LIN {X 0,Y 523.661,Z 782.836,A -85,B 0,C 180,E1 -4887.396,E2 -4887.396} C_VEL
LIN {X 0,Y 523.608,Z 785.881,A -85,B 0,C 180,E1 -4887.924,E2 -4887.924} C_VEL
LIN {X 0,Y 522.919,Z 788.862,A -85,B 0,C 180,E1 -4888.477,E2 -4888.477} C_VEL
LIN {X 0,Y 519.953,Z 793.273,A -85,B 0,C 180,E1 -4889.399,E2 -4889.399} C_VEL
LIN {X 0,Y 516.983,Z 796.944,A -85,B 0,C 180,E1 -4890.367,E2 -4890.367} C_VEL
LIN {X 0,Y 516.299,Z 798.763,A -85,B 0,C 180,E1 -4890.988,E2 -4890.988} C_VEL
LIN {X 0,Y 516.19,Z 801.916,A -85,B 0,C 180,E1 -4892.422,E2 -4892.422} C_VEL
LIN {X 0,Y 516.167,Z 803.743,A -85,B 0,C 180,E1 -4893.934,E2 -4893.934} C_VEL
LIN {X 0,Y 516.163,Z 804.121,A -85,B 0,C 180,E1 -4895.221,E2 -4895.221} C_VEL
LIN {X 0,Y 516.15,Z 803.144,A -85,B 0,C 180,E1 -4896.806,E2 -4896.806} C_VEL
LIN {X 0,Y 516.166,Z 801.549,A -85,B 0,C 180,E1 -4897.843,E2 -4897.843} C_VEL
LIN {X 0,Y 516.284,Z 798.724,A -85,B 0,C 180,E1 -4899.113,E2 -4899.113} C_VEL
LIN {X 0,Y 516.35,Z 794.83,A -85,B 0,C 180,E1 -4900.342,E2 -4900.342} C_VEL
LIN {X 0,Y 516.401,Z 789.867,A -85,B 0,C 180,E1 -4901.539,E2 -4901.539} C_VEL
LIN {X 0,Y 516.631,Z 782.827,A -85,B 0,C 180,E1 -4902.857,E2 -4902.857} C_VEL
LIN {X 0,Y 516.794,Z 775.836,A -85,B 0,C 180,E1 -4903.913,E2 -4903.913} C_VEL
LIN {X 0,Y 517.07,Z 766.749,A -85,B 0,C 180,E1 -4905.028,E2 -4905.028} C_VEL
LIN {X 0,Y 517.366,Z 756.345,A -85,B 0,C 180,E1 -4906.051,E2 -4906.051} C_VEL
LIN {X 0,Y 517.663,Z 745.961,A -85,B 0,C 180,E1 -4906.873,E2 -4906.873} C_VEL
LIN {X 0,Y 517.987,Z 734.619,A -85,B 0,C 180,E1 -4907.583,E2 -4907.583} C_VEL
LIN {X 0,Y 518.283,Z 722.652,A -85,B 0,C 180,E1 -4908.16,E2 -4908.16} C_VEL
LIN {X 0,Y 518.465,Z 709.924,A -85,B 0,C 180,E1 -4908.604,E2 -4908.604} C_VEL
LIN {X 0,Y 518.673,Z 696.818,A -85,B 0,C 180,E1 -4908.89,E2 -4908.89} C_VEL
LIN {X 0,Y 518.951,Z 604.587,A -85,B 0,C 180,E1 -4910.186,E2 -4910.186} C_VEL
LIN {X 0,Y 517.134,Z 594.704,A -85,B 0,C 180,E1 -4910.404,E2 -4910.404} C_VEL
LIN {X 0,Y 517.332,Z 583.642,A -85,B 0,C 180,E1 -4912.806,E2 -4912.806} C_VEL
LIN {X 0,Y 516.951,Z 581.095,A -85,B 0,C 180,E1 -4913.399,E2 -4913.399} C_VEL
LIN {X 0,Y 516.911,Z 581.098,A -85,B 0,C 180,E1 -4916.122,E2 -4916.122} C_VEL
LIN {X 0,Y 516.887,Z 581.094,A -85,B 0,C 180,E1 -4918.937,E2 -4918.937} C_VEL
LIN {X 0,Y 516.917,Z 581.093,A -85,B 0,C 180,E1 -4921.586,E2 -4921.586} C_VEL
LIN {X 0,Y 516.929,Z 581.096,A -85,B 0,C 180,E1 -4924.212,E2 -4924.212} C_VEL
LIN {X 0,Y 516.87,Z 581.097,A -85,B 0,C 180,E1 -4926.778,E2 -4926.778} C_VEL
LIN {X 0,Y 516.938,Z 581.09,A -85,B 0,C 180,E1 -4929.732,E2 -4929.732} C_VEL
LIN {X 0,Y 516.931,Z 581.092,A -85,B 0,C 180,E1 -4932.597,E2 -4932.597} C_VEL
LIN {X 0,Y 516.942,Z 581.087,A -85,B 0,C 180,E1 -4935.031,E2 -4935.031} C_VEL
LIN {X 0,Y 517.005,Z 581.087,A -85,B 0,C 180,E1 -4938.236,E2 -4938.236} C_VEL
LIN {X 0,Y 516.969,Z 581.083,A -85,B 0,C 180,E1 -4941.401,E2 -4941.401} C_VEL
LIN {X 0,Y 517.011,Z 581.079,A -85,B 0,C 180,E1 -4943.758,E2 -4943.758} C_VEL
LIN {X 0,Y 517.086,Z 581.069,A -85,B 0,C 180,E1 -4947.664,E2 -4947.664} C_VEL
LIN {X 0,Y 517.095,Z 581.074,A -85,B 0,C 180,E1 -4950.78,E2 -4950.78} C_VEL
LIN {X 0,Y 517.016,Z 581.08,A -85,B 0,C 180,E1 -4953.118,E2 -4953.118} C_VEL
LIN {X 0,Y 517.012,Z 581.081,A -85,B 0,C 180,E1 -4956.244,E2 -4956.244} C_VEL
LIN {X 0,Y 516.957,Z 581.086,A -85,B 0,C 180,E1 -4959.39,E2 -4959.39} C_VEL
LIN {X 0,Y 516.956,Z 581.085,A -85,B 0,C 180,E1 -4961.808,E2 -4961.808} C_VEL
LIN {X 0,Y 516.948,Z 581.09,A -85,B 0,C 180,E1 -4965.147,E2 -4965.147} C_VEL
LIN {X 0,Y 516.928,Z 581.089,A -85,B 0,C 180,E1 -4968.223,E2 -4968.223} C_VEL
LIN {X 0,Y 516.916,Z 581.096,A -85,B 0,C 180,E1 -4970.702,E2 -4970.702} C_VEL
LIN {X 0,Y 516.906,Z 581.091,A -85,B 0,C 180,E1 -4974.073,E2 -4974.073} C_VEL
LIN {X 0,Y 516.93,Z 581.092,A -85,B 0,C 180,E1 -4976.658,E2 -4976.658} C_VEL
LIN {X 0,Y 516.915,Z 581.093,A -85,B 0,C 180,E1 -4979.524,E2 -4979.524} C_VEL
LIN {X 0,Y 516.899,Z 581.094,A -85,B 0,C 180,E1 -4982.544,E2 -4982.544} C_VEL
LIN {X 0,Y 516.874,Z 581.103,A -85,B 0,C 180,E1 -4985.331,E2 -4985.331} C_VEL
LIN {X 0,Y 516.885,Z 581.095,A -85,B 0,C 180,E1 -4987.944,E2 -4987.944} C_VEL
LIN {X 0,Y 516.887,Z 581.095,A -85,B 0,C 180,E1 -4990.742,E2 -4990.742} C_VEL
LIN {X 0,Y 516.886,Z 581.096,A -85,B 0,C 180,E1 -4992.832,E2 -4992.832} C_VEL
LIN {X 0,Y 516.899,Z 581.096,A -85,B 0,C 180,E1 -4995.007,E2 -4995.007} C_VEL
LIN {X 0,Y 516.919,Z 581.089,A -85,B 0,C 180,E1 -4998.399,E2 -4998.399} C_VEL
LIN {X 0,Y 516.885,Z 581.1,A -85,B 0,C 180,E1 -5001.285,E2 -5001.285} C_VEL
LIN {X 0,Y 516.875,Z 581.096,A -85,B 0,C 180,E1 -5004.22,E2 -5004.22} C_VEL
LIN {X 0,Y 516.899,Z 581.094,A -85,B 0,C 180,E1 -5007.053,E2 -5007.053} C_VEL
LIN {X 0,Y 516.897,Z 581.099,A -85,B 0,C 180,E1 -5009.797,E2 -5009.797} C_VEL
LIN {X 0,Y 516.931,Z 581.088,A -85,B 0,C 180,E1 -5012.468,E2 -5012.468} C_VEL
LIN {X 0,Y 516.88,Z 581.095,A -85,B 0,C 180,E1 -5015.07,E2 -5015.07} C_VEL
LIN {X 0,Y 516.873,Z 581.102,A -85,B 0,C 180,E1 -5017.622,E2 -5017.622} C_VEL
LIN {X 0,Y 516.936,Z 581.092,A -85,B 0,C 180,E1 -5020.13,E2 -5020.13} C_VEL
LIN {X 0,Y 516.912,Z 581.091,A -85,B 0,C 180,E1 -5022.596,E2 -5022.596} C_VEL
LIN {X 0,Y 516.948,Z 581.086,A -85,B 0,C 180,E1 -5025.03,E2 -5025.03} C_VEL
LIN {X 0,Y 516.971,Z 581.089,A -85,B 0,C 180,E1 -5028.234,E2 -5028.234} C_VEL
LIN {X 0,Y 516.97,Z 581.084,A -85,B 0,C 180,E1 -5031.4,E2 -5031.4} C_VEL
LIN {X 0,Y 517.015,Z 581.082,A -85,B 0,C 180,E1 -5033.757,E2 -5033.757} C_VEL
LIN {X 0,Y 517.089,Z 581.071,A -85,B 0,C 180,E1 -5037.663,E2 -5037.663} C_VEL
LIN {X 0,Y 517.098,Z 581.069,A -85,B 0,C 180,E1 -5040.779,E2 -5040.779} C_VEL
LIN {X 0,Y 517.017,Z 581.077,A -85,B 0,C 180,E1 -5043.117,E2 -5043.117} C_VEL
LIN {X 0,Y 517.014,Z 581.087,A -85,B 0,C 180,E1 -5046.243,E2 -5046.243} C_VEL
LIN {X 0,Y 516.95,Z 581.086,A -85,B 0,C 180,E1 -5049.389,E2 -5049.389} C_VEL
LIN {X 0,Y 516.958,Z 581.086,A -85,B 0,C 180,E1 -5051.807,E2 -5051.807} C_VEL
LIN {X 0,Y 516.95,Z 581.087,A -85,B 0,C 180,E1 -5055.146,E2 -5055.146} C_VEL
LIN {X 0,Y 516.922,Z 581.094,A -85,B 0,C 180,E1 -5058.222,E2 -5058.222} C_VEL
LIN {X 0,Y 516.918,Z 581.097,A -85,B 0,C 180,E1 -5060.701,E2 -5060.701} C_VEL
LIN {X 0,Y 516.908,Z 581.093,A -85,B 0,C 180,E1 -5064.072,E2 -5064.072} C_VEL
LIN {X 0,Y 516.929,Z 581.098,A -85,B 0,C 180,E1 -5066.658,E2 -5066.658} C_VEL
LIN {X 0,Y 516.916,Z 581.09,A -85,B 0,C 180,E1 -5069.524,E2 -5069.524} C_VEL
LIN {X 0,Y 516.901,Z 581.098,A -85,B 0,C 180,E1 -5072.543,E2 -5072.543} C_VEL
LIN {X 0,Y 516.874,Z 581.098,A -85,B 0,C 180,E1 -5075.33,E2 -5075.33} C_VEL
LIN {X 0,Y 516.886,Z 581.094,A -85,B 0,C 180,E1 -5077.943,E2 -5077.943} C_VEL
LIN {X 0,Y 516.89,Z 581.1,A -85,B 0,C 180,E1 -5080.741,E2 -5080.741} C_VEL
LIN {X 0,Y 516.89,Z 581.101,A -85,B 0,C 180,E1 -5082.831,E2 -5082.831} C_VEL
LIN {X 0,Y 516.929,Z 581.098,A -85,B 0,C 180,E1 -5085.01,E2 -5085.01} C_VEL
LIN {X 0,Y 516.919,Z 581.091,A -85,B 0,C 180,E1 -5088.398,E2 -5088.398} C_VEL
LIN {X 0,Y 516.887,Z 581.101,A -85,B 0,C 180,E1 -5091.284,E2 -5091.284} C_VEL
LIN {X 0,Y 516.878,Z 581.095,A -85,B 0,C 180,E1 -5094.219,E2 -5094.219} C_VEL
LIN {X 0,Y 516.902,Z 581.1,A -85,B 0,C 180,E1 -5097.053,E2 -5097.053} C_VEL
LIN {X 0,Y 516.892,Z 581.097,A -85,B 0,C 180,E1 -5099.796,E2 -5099.796} C_VEL
LIN {X 0,Y 516.931,Z 581.091,A -85,B 0,C 180,E1 -5102.467,E2 -5102.467} C_VEL
LIN {X 0,Y 516.962,Z 581.168,A -85,B 0,C 180,E1 -5104.186,E2 -5104.186} C_VEL
LIN {X 0,Y 518.877,Z 591.241,A -85,B 0,C 180,E1 -5105.833,E2 -5105.833} C_VEL
LIN {X 0,Y 518.458,Z 607.819,A -85,B 0,C 180,E1 -5108.321,E2 -5108.321} C_VEL
LIN {X 0,Y 517.951,Z 628.652,A -85,B 0,C 180,E1 -5111.405,E2 -5111.405} C_VEL
LIN {X 0,Y 517.414,Z 650.625,A -85,B 0,C 180,E1 -5114.621,E2 -5114.621} C_VEL
LIN {X 0,Y 519.067,Z 662.608,A -85,B 0,C 180,E1 -5114.855,E2 -5114.855} C_VEL
LIN {X 0,Y 518.619,Z 760.064,A -85,B 0,C 180,E1 -5116.231,E2 -5116.231} C_VEL
LIN {X 0,Y 518.39,Z 773.157,A -85,B 0,C 180,E1 -5116.574,E2 -5116.574} C_VEL
LIN {X 0,Y 518.11,Z 785.812,A -85,B 0,C 180,E1 -5117.066,E2 -5117.066} C_VEL
LIN {X 0,Y 517.849,Z 797.67,A -85,B 0,C 180,E1 -5117.694,E2 -5117.694} C_VEL
LIN {X 0,Y 517.502,Z 810.055,A -85,B 0,C 180,E1 -5118.543,E2 -5118.543} C_VEL
LIN {X 0,Y 517.194,Z 820.324,A -85,B 0,C 180,E1 -5119.429,E2 -5119.429} C_VEL
LIN {X 0,Y 516.94,Z 829.561,A -85,B 0,C 180,E1 -5120.412,E2 -5120.412} C_VEL
LIN {X 0,Y 516.716,Z 838.56,A -85,B 0,C 180,E1 -5121.592,E2 -5121.592} C_VEL
LIN {X 0,Y 516.511,Z 845.802,A -85,B 0,C 180,E1 -5122.769,E2 -5122.769} C_VEL
LIN {X 0,Y 516.427,Z 850.672,A -85,B 0,C 180,E1 -5123.749,E2 -5123.749} C_VEL
LIN {X 0,Y 516.314,Z 855.37,A -85,B 0,C 180,E1 -5124.923,E2 -5124.923} C_VEL
LIN {X 0,Y 516.355,Z 858.955,A -85,B 0,C 180,E1 -5126.097,E2 -5126.097} C_VEL
LIN {X 0,Y 516.283,Z 860.805,A -85,B 0,C 180,E1 -5126.878,E2 -5126.878} C_VEL
LIN {X 0,Y 516.26,Z 862.191,A -85,B 0,C 180,E1 -5127.659,E2 -5127.659} C_VEL
LIN {X 0,Y 516.16,Z 863.785,A -85,B 0,C 180,E1 -5129.219,E2 -5129.219} C_VEL
LIN {X 0,Y 516.154,Z 864,A -85,B 0,C 180,E1 -5129.999,E2 -5129.999} C_VEL
LIN {X 0,Y 516.191,Z 863.184,A -85,B 0,C 180,E1 -5131.56,E2 -5131.56} C_VEL
LIN {X 0,Y 516.26,Z 862.197,A -85,B 0,C 180,E1 -5132.34,E2 -5132.34} C_VEL
LIN {X 0,Y 516.282,Z 860.812,A -85,B 0,C 180,E1 -5133.12,E2 -5133.12} C_VEL
LIN {X 0,Y 516.344,Z 857.897,A -85,B 0,C 180,E1 -5134.292,E2 -5134.292} C_VEL
LIN {X 0,Y 516.405,Z 853.951,A -85,B 0,C 180,E1 -5135.466,E2 -5135.466} C_VEL
LIN {X 0,Y 516.479,Z 848.069,A -85,B 0,C 180,E1 -5136.797,E2 -5136.797} C_VEL
LIN {X 0,Y 516.64,Z 841.144,A -85,B 0,C 180,E1 -5138.014,E2 -5138.014} C_VEL
LIN {X 0,Y 516.844,Z 832.801,A -85,B 0,C 180,E1 -5139.193,E2 -5139.193} C_VEL
LIN {X 0,Y 517.072,Z 824.246,A -85,B 0,C 180,E1 -5140.176,E2 -5140.176} C_VEL
LIN {X 0,Y 517.432,Z 813.681,A -85,B 0,C 180,E1 -5141.159,E2 -5141.159} C_VEL
LIN {X 0,Y 517.704,Z 803.398,A -85,B 0,C 180,E1 -5141.935,E2 -5141.935} C_VEL
LIN {X 0,Y 518.016,Z 791.756,A -85,B 0,C 180,E1 -5142.636,E2 -5142.636} C_VEL
LIN {X 0,Y 518.272,Z 779.951,A -85,B 0,C 180,E1 -5143.178,E2 -5143.178} C_VEL
LIN {X 0,Y 518.472,Z 766.341,A -85,B 0,C 180,E1 -5143.621,E2 -5143.621} C_VEL
LIN {X 0,Y 518.646,Z 752.686,A -85,B 0,C 180,E1 -5143.892,E2 -5143.892} C_VEL
LIN {X 0,Y 518.905,Z 660.251,A -85,B 0,C 180,E1 -5145.177,E2 -5145.177} C_VEL
LIN {X 0,Y 517.401,Z 650.463,A -85,B 0,C 180,E1 -5145.372,E2 -5145.372} C_VEL
LIN {X 0,Y 517.889,Z 628.311,A -85,B 0,C 180,E1 -5148.596,E2 -5148.596} C_VEL
LIN {X 0,Y 518.387,Z 608.713,A -85,B 0,C 180,E1 -5151.471,E2 -5151.471} C_VEL
LIN {X 0,Y 518.791,Z 590.699,A -85,B 0,C 180,E1 -5154.165,E2 -5154.165} C_VEL
LIN {X 0,Y 516.953,Z 581.093,A -85,B 0,C 180,E1 -5155.733,E2 -5155.733} C_VEL
LIN {X 0,Y 516.918,Z 581.099,A -85,B 0,C 180,E1 -5158.414,E2 -5158.414} C_VEL
LIN {X 0,Y 516.887,Z 581.1,A -85,B 0,C 180,E1 -5161.108,E2 -5161.108} C_VEL
LIN {X 0,Y 516.91,Z 581.095,A -85,B 0,C 180,E1 -5163.966,E2 -5163.966} C_VEL
LIN {X 0,Y 516.88,Z 581.102,A -85,B 0,C 180,E1 -5166.745,E2 -5166.745} C_VEL
LIN {X 0,Y 516.9,Z 581.095,A -85,B 0,C 180,E1 -5169.718,E2 -5169.718} C_VEL
LIN {X 0,Y 516.915,Z 581.094,A -85,B 0,C 180,E1 -5171.773,E2 -5171.773} C_VEL
LIN {X 0,Y 516.918,Z 581.094,A -85,B 0,C 180,E1 -5175.009,E2 -5175.009} C_VEL
LIN {X 0,Y 516.918,Z 581.099,A -85,B 0,C 180,E1 -5178.397,E2 -5178.397} C_VEL
LIN {X 0,Y 516.904,Z 581.092,A -85,B 0,C 180,E1 -5181.286,E2 -5181.286} C_VEL
LIN {X 0,Y 516.885,Z 581.099,A -85,B 0,C 180,E1 -5184.221,E2 -5184.221} C_VEL
LIN {X 0,Y 516.892,Z 581.095,A -85,B 0,C 180,E1 -5187.053,E2 -5187.053} C_VEL
LIN {X 0,Y 516.896,Z 581.094,A -85,B 0,C 180,E1 -5189.796,E2 -5189.796} C_VEL
LIN {X 0,Y 516.923,Z 581.098,A -85,B 0,C 180,E1 -5192.467,E2 -5192.467} C_VEL
LIN {X 0,Y 516.905,Z 581.093,A -85,B 0,C 180,E1 -5195.071,E2 -5195.071} C_VEL
LIN {X 0,Y 516.879,Z 581.103,A -85,B 0,C 180,E1 -5198.462,E2 -5198.462} C_VEL
LIN {X 0,Y 516.897,Z 581.095,A -85,B 0,C 180,E1 -5200.955,E2 -5200.955} C_VEL
LIN {X 0,Y 516.908,Z 581.092,A -85,B 0,C 180,E1 -5203.41,E2 -5203.41} C_VEL
LIN {X 0,Y 516.888,Z 581.095,A -85,B 0,C 180,E1 -5205.833,E2 -5205.833} C_VEL
LIN {X 0,Y 516.996,Z 581.087,A -85,B 0,C 180,E1 -5208.234,E2 -5208.234} C_VEL
LIN {X 0,Y 516.964,Z 581.085,A -85,B 0,C 180,E1 -5211.399,E2 -5211.399} C_VEL
LIN {X 0,Y 517.002,Z 581.082,A -85,B 0,C 180,E1 -5213.757,E2 -5213.757} C_VEL
LIN {X 0,Y 517.076,Z 581.072,A -85,B 0,C 180,E1 -5217.663,E2 -5217.663} C_VEL
LIN {X 0,Y 517.087,Z 581.073,A -85,B 0,C 180,E1 -5220.779,E2 -5220.779} C_VEL
LIN {X 0,Y 517.009,Z 581.081,A -85,B 0,C 180,E1 -5223.117,E2 -5223.117} C_VEL
LIN {X 0,Y 517.007,Z 581.089,A -85,B 0,C 180,E1 -5226.243,E2 -5226.243} C_VEL
LIN {X 0,Y 516.951,Z 581.088,A -85,B 0,C 180,E1 -5229.389,E2 -5229.389} C_VEL
LIN {X 0,Y 516.975,Z 581.087,A -85,B 0,C 180,E1 -5231.824,E2 -5231.824} C_VEL
LIN {X 0,Y 516.922,Z 581.097,A -85,B 0,C 180,E1 -5235.141,E2 -5235.141} C_VEL
LIN {X 0,Y 516.987,Z 581.184,A -85,B 0,C 180,E1 -5236.638,E2 -5236.638} C_VEL
LIN {X 0,Y 517.37,Z 585.996,A -85,B 0,C 180,E1 -5237.711,E2 -5237.711} C_VEL
LIN {X 0,Y 517.11,Z 595.183,A -85,B 0,C 180,E1 -5239.708,E2 -5239.708} C_VEL
LIN {X 0,Y 519.115,Z 606.073,A -85,B 0,C 180,E1 -5239.927,E2 -5239.927} C_VEL
LIN {X 0,Y 518.62,Z 701.328,A -85,B 0,C 180,E1 -5241.28,E2 -5241.28} C_VEL
LIN {X 0,Y 518.403,Z 714.472,A -85,B 0,C 180,E1 -5241.628,E2 -5241.628} C_VEL
LIN {X 0,Y 518.174,Z 726.854,A -85,B 0,C 180,E1 -5242.109,E2 -5242.109} C_VEL
LIN {X 0,Y 517.881,Z 739.146,A -85,B 0,C 180,E1 -5242.766,E2 -5242.766} C_VEL
LIN {X 0,Y 517.582,Z 749.94,A -85,B 0,C 180,E1 -5243.507,E2 -5243.507} C_VEL
LIN {X 0,Y 517.235,Z 760.82,A -85,B 0,C 180,E1 -5244.446,E2 -5244.446} C_VEL
LIN {X 0,Y 516.994,Z 769.357,A -85,B 0,C 180,E1 -5245.354,E2 -5245.354} C_VEL
LIN {X 0,Y 516.753,Z 777.316,A -85,B 0,C 180,E1 -5246.378,E2 -5246.378} C_VEL
LIN {X 0,Y 516.575,Z 784.742,A -85,B 0,C 180,E1 -5247.553,E2 -5247.553} C_VEL
LIN {X 0,Y 516.441,Z 791.385,A -85,B 0,C 180,E1 -5248.888,E2 -5248.888} C_VEL
LIN {X 0,Y 516.32,Z 796.553,A -85,B 0,C 180,E1 -5250.241,E2 -5250.241} C_VEL
LIN {X 0,Y 516.299,Z 798.763,A -85,B 0,C 180,E1 -5250.988,E2 -5250.988} C_VEL
LIN {X 0,Y 515.62,Z 800.372,A -85,B 0,C 180,E1 -5251.615,E2 -5251.615} C_VEL
LIN {X 0,Y 512.675,Z 802.519,A -85,B 0,C 180,E1 -5252.642,E2 -5252.642} C_VEL
LIN {X 0,Y 510.201,Z 803.709,A -85,B 0,C 180,E1 -5253.48,E2 -5253.48} C_VEL
LIN {X 0,Y 509.161,Z 804.278,A -85,B 0,C 180,E1 -5254.132,E2 -5254.132} C_VEL
LIN {X 0,Y 509.09,Z 804.395,A -85,B 0,C 180,E1 -5254.354,E2 -5254.354} C_VEL
LIN {X 0,Y 509.079,Z 804.487,A -85,B 0,C 180,E1 -5255.463,E2 -5255.463} C_VEL
LIN {X 0,Y 509.063,Z 803.579,A -85,B 0,C 180,E1 -5256.802,E2 -5256.802} C_VEL
LIN {X 0,Y 509.096,Z 801.528,A -85,B 0,C 180,E1 -5258.107,E2 -5258.107} C_VEL
LIN {X 0,Y 509.228,Z 798.463,A -85,B 0,C 180,E1 -5259.41,E2 -5259.41} C_VEL
LIN {X 0,Y 509.291,Z 794.427,A -85,B 0,C 180,E1 -5260.628,E2 -5260.628} C_VEL
LIN {X 0,Y 509.38,Z 789.237,A -85,B 0,C 180,E1 -5261.839,E2 -5261.839} C_VEL
LIN {X 0,Y 509.602,Z 782.773,A -85,B 0,C 180,E1 -5263.037,E2 -5263.037} C_VEL
LIN {X 0,Y 509.812,Z 774.925,A -85,B 0,C 180,E1 -5264.207,E2 -5264.207} C_VEL
LIN {X 0,Y 510.159,Z 765.221,A -85,B 0,C 180,E1 -5265.367,E2 -5265.367} C_VEL
LIN {X 0,Y 510.447,Z 755.678,A -85,B 0,C 180,E1 -5266.289,E2 -5266.289} C_VEL
LIN {X 0,Y 510.772,Z 744.089,A -85,B 0,C 180,E1 -5267.185,E2 -5267.185} C_VEL
LIN {X 0,Y 511.114,Z 733.272,A -85,B 0,C 180,E1 -5267.844,E2 -5267.844} C_VEL
LIN {X 0,Y 511.438,Z 720.697,A -85,B 0,C 180,E1 -5268.427,E2 -5268.427} C_VEL
LIN {X 0,Y 511.625,Z 707.479,A -85,B 0,C 180,E1 -5268.858,E2 -5268.858} C_VEL
LIN {X 0,Y 511.816,Z 695.004,A -85,B 0,C 180,E1 -5269.108,E2 -5269.108} C_VEL
LIN {X 0,Y 512.143,Z 605.61,A -85,B 0,C 180,E1 -5270.382,E2 -5270.382} C_VEL
LIN {X 0,Y 510.163,Z 595.045,A -85,B 0,C 180,E1 -5270.621,E2 -5270.621} C_VEL
LIN {X 0,Y 510.383,Z 585.504,A -85,B 0,C 180,E1 -5272.709,E2 -5272.709} C_VEL
LIN {X 0,Y 509.909,Z 581.973,A -85,B 0,C 180,E1 -5273.55,E2 -5273.55} C_VEL
LIN {X 0,Y 509.86,Z 581.972,A -85,B 0,C 180,E1 -5276.54,E2 -5276.54} C_VEL
LIN {X 0,Y 509.842,Z 581.973,A -85,B 0,C 180,E1 -5279.335,E2 -5279.335} C_VEL
LIN {X 0,Y 509.892,Z 581.974,A -85,B 0,C 180,E1 -5282.056,E2 -5282.056} C_VEL
LIN {X 0,Y 509.875,Z 581.968,A -85,B 0,C 180,E1 -5284.705,E2 -5284.705} C_VEL
LIN {X 0,Y 509.835,Z 581.973,A -85,B 0,C 180,E1 -5287.456,E2 -5287.456} C_VEL
LIN {X 0,Y 509.916,Z 581.966,A -85,B 0,C 180,E1 -5289.846,E2 -5289.846} C_VEL
LIN {X 0,Y 509.886,Z 581.966,A -85,B 0,C 180,E1 -5293.176,E2 -5293.176} C_VEL
LIN {X 0,Y 509.865,Z 581.969,A -85,B 0,C 180,E1 -5295.635,E2 -5295.635} C_VEL
LIN {X 0,Y 509.923,Z 581.963,A -85,B 0,C 180,E1 -5298.876,E2 -5298.876} C_VEL
LIN {X 0,Y 509.952,Z 581.962,A -85,B 0,C 180,E1 -5302.079,E2 -5302.079} C_VEL
LIN {X 0,Y 509.982,Z 581.963,A -85,B 0,C 180,E1 -5304.465,E2 -5304.465} C_VEL
LIN {X 0,Y 510.057,Z 581.944,A -85,B 0,C 180,E1 -5307.632,E2 -5307.632} C_VEL
LIN {X 0,Y 510.066,Z 581.949,A -85,B 0,C 180,E1 -5310.79,E2 -5310.79} C_VEL
LIN {X 0,Y 509.958,Z 581.958,A -85,B 0,C 180,E1 -5313.161,E2 -5313.161} C_VEL
LIN {X 0,Y 509.981,Z 581.958,A -85,B 0,C 180,E1 -5316.33,E2 -5316.33} C_VEL
LIN {X 0,Y 509.919,Z 581.971,A -85,B 0,C 180,E1 -5318.721,E2 -5318.721} C_VEL
LIN {X 0,Y 509.908,Z 581.963,A -85,B 0,C 180,E1 -5321.932,E2 -5321.932} C_VEL
LIN {X 0,Y 509.897,Z 581.968,A -85,B 0,C 180,E1 -5325.242,E2 -5325.242} C_VEL
LIN {X 0,Y 509.885,Z 581.966,A -85,B 0,C 180,E1 -5327.999,E2 -5327.999} C_VEL
LIN {X 0,Y 509.854,Z 581.978,A -85,B 0,C 180,E1 -5331.002,E2 -5331.002} C_VEL
LIN {X 0,Y 509.867,Z 581.97,A -85,B 0,C 180,E1 -5334.427,E2 -5334.427} C_VEL
LIN {X 0,Y 509.889,Z 581.975,A -85,B 0,C 180,E1 -5337.056,E2 -5337.056} C_VEL
LIN {X 0,Y 509.861,Z 581.97,A -85,B 0,C 180,E1 -5339.752,E2 -5339.752} C_VEL
LIN {X 0,Y 509.877,Z 581.971,A -85,B 0,C 180,E1 -5342.775,E2 -5342.775} C_VEL
LIN {X 0,Y 509.833,Z 581.976,A -85,B 0,C 180,E1 -5345.579,E2 -5345.579} C_VEL
LIN {X 0,Y 509.855,Z 581.97,A -85,B 0,C 180,E1 -5348.338,E2 -5348.338} C_VEL
LIN {X 0,Y 509.859,Z 581.977,A -85,B 0,C 180,E1 -5351.426,E2 -5351.426} C_VEL
LIN {X 0,Y 509.843,Z 581.972,A -85,B 0,C 180,E1 -5354.67,E2 -5354.67} C_VEL
LIN {X 0,Y 509.839,Z 581.98,A -85,B 0,C 180,E1 -5357.511,E2 -5357.511} C_VEL
LIN {X 0,Y 509.85,Z 581.97,A -85,B 0,C 180,E1 -5360.648,E2 -5360.648} C_VEL
LIN {X 0,Y 509.829,Z 581.98,A -85,B 0,C 180,E1 -5363.647,E2 -5363.647} C_VEL
LIN {X 0,Y 509.863,Z 581.968,A -85,B 0,C 180,E1 -5366.539,E2 -5366.539} C_VEL
LIN {X 0,Y 509.85,Z 581.975,A -85,B 0,C 180,E1 -5369.335,E2 -5369.335} C_VEL
LIN {X 0,Y 509.897,Z 581.968,A -85,B 0,C 180,E1 -5372.055,E2 -5372.055} C_VEL
LIN {X 0,Y 509.845,Z 581.971,A -85,B 0,C 180,E1 -5374.702,E2 -5374.702} C_VEL
LIN {X 0,Y 509.831,Z 581.977,A -85,B 0,C 180,E1 -5377.458,E2 -5377.458} C_VEL
LIN {X 0,Y 509.922,Z 581.971,A -85,B 0,C 180,E1 -5379.845,E2 -5379.845} C_VEL
LIN {X 0,Y 509.879,Z 581.967,A -85,B 0,C 180,E1 -5383.175,E2 -5383.175} C_VEL
LIN {X 0,Y 509.869,Z 581.973,A -85,B 0,C 180,E1 -5385.634,E2 -5385.634} C_VEL
LIN {X 0,Y 509.918,Z 581.962,A -85,B 0,C 180,E1 -5388.875,E2 -5388.875} C_VEL
LIN {X 0,Y 509.956,Z 581.966,A -85,B 0,C 180,E1 -5392.079,E2 -5392.079} C_VEL
LIN {X 0,Y 509.986,Z 581.957,A -85,B 0,C 180,E1 -5394.464,E2 -5394.464} C_VEL
LIN {X 0,Y 510.06,Z 581.946,A -85,B 0,C 180,E1 -5397.631,E2 -5397.631} C_VEL
LIN {X 0,Y 510.069,Z 581.945,A -85,B 0,C 180,E1 -5400.79,E2 -5400.79} C_VEL
LIN {X 0,Y 509.959,Z 581.956,A -85,B 0,C 180,E1 -5403.16,E2 -5403.16} C_VEL
LIN {X 0,Y 509.982,Z 581.963,A -85,B 0,C 180,E1 -5406.33,E2 -5406.33} C_VEL
LIN {X 0,Y 509.917,Z 581.966,A -85,B 0,C 180,E1 -5408.72,E2 -5408.72} C_VEL
LIN {X 0,Y 509.91,Z 581.965,A -85,B 0,C 180,E1 -5411.932,E2 -5411.932} C_VEL
LIN {X 0,Y 509.9,Z 581.964,A -85,B 0,C 180,E1 -5415.242,E2 -5415.242} C_VEL
LIN {X 0,Y 509.873,Z 581.969,A -85,B 0,C 180,E1 -5417.993,E2 -5417.993} C_VEL
LIN {X 0,Y 509.892,Z 581.972,A -85,B 0,C 180,E1 -5420.401,E2 -5420.401} C_VEL
LIN {X 0,Y 509.835,Z 581.972,A -85,B 0,C 180,E1 -5423.563,E2 -5423.563} C_VEL
LIN {X 0,Y 509.916,Z 581.967,A -85,B 0,C 180,E1 -5426.378,E2 -5426.378} C_VEL
LIN {X 0,Y 509.882,Z 581.974,A -85,B 0,C 180,E1 -5428.844,E2 -5428.844} C_VEL
LIN {X 0,Y 509.825,Z 581.973,A -85,B 0,C 180,E1 -5431.59,E2 -5431.59} C_VEL
LIN {X 0,Y 509.855,Z 581.973,A -85,B 0,C 180,E1 -5434.413,E2 -5434.413} C_VEL
LIN {X 0,Y 509.822,Z 581.976,A -85,B 0,C 180,E1 -5437.341,E2 -5437.341} C_VEL
LIN {X 0,Y 509.844,Z 581.973,A -85,B 0,C 180,E1 -5440.382,E2 -5440.382} C_VEL
LIN {X 0,Y 509.83,Z 581.981,A -85,B 0,C 180,E1 -5443.062,E2 -5443.062} C_VEL
LIN {X 0,Y 509.836,Z 581.972,A -85,B 0,C 180,E1 -5445.792,E2 -5445.792} C_VEL
LIN {X 0,Y 509.861,Z 581.971,A -85,B 0,C 180,E1 -5448.574,E2 -5448.574} C_VEL
LIN {X 0,Y 509.856,Z 581.97,A -85,B 0,C 180,E1 -5451.786,E2 -5451.786} C_VEL
LIN {X 0,Y 509.838,Z 581.973,A -85,B 0,C 180,E1 -5454.622,E2 -5454.622} C_VEL
LIN {X 0,Y 509.869,Z 581.975,A -85,B 0,C 180,E1 -5457.481,E2 -5457.481} C_VEL
LIN {X 0,Y 509.863,Z 581.971,A -85,B 0,C 180,E1 -5460.273,E2 -5460.273} C_VEL
LIN {X 0,Y 509.889,Z 581.973,A -85,B 0,C 180,E1 -5462.944,E2 -5462.944} C_VEL
LIN {X 0,Y 509.917,Z 582.08,A -85,B 0,C 180,E1 -5463.994,E2 -5463.994} C_VEL
LIN {X 0,Y 511.907,Z 592.172,A -85,B 0,C 180,E1 -5465.677,E2 -5465.677} C_VEL
LIN {X 0,Y 511.666,Z 604.697,A -85,B 0,C 180,E1 -5467.594,E2 -5467.594} C_VEL
LIN {X 0,Y 511.054,Z 625.542,A -85,B 0,C 180,E1 -5470.728,E2 -5470.728} C_VEL
LIN {X 0,Y 510.506,Z 646.255,A -85,B 0,C 180,E1 -5473.812,E2 -5473.812} C_VEL
LIN {X 0,Y 510.36,Z 650.353,A -85,B 0,C 180,E1 -5474.419,E2 -5474.419} C_VEL
LIN {X 0,Y 512.19,Z 662.783,A -85,B 0,C 180,E1 -5474.658,E2 -5474.658} C_VEL
LIN {X 0,Y 511.706,Z 759.346,A -85,B 0,C 180,E1 -5476.041,E2 -5476.041} C_VEL
LIN {X 0,Y 511.43,Z 773.304,A -85,B 0,C 180,E1 -5476.414,E2 -5476.414} C_VEL
LIN {X 0,Y 511.142,Z 786.318,A -85,B 0,C 180,E1 -5476.937,E2 -5476.937} C_VEL
LIN {X 0,Y 510.836,Z 798.226,A -85,B 0,C 180,E1 -5477.59,E2 -5477.59} C_VEL
LIN {X 0,Y 510.494,Z 809.562,A -85,B 0,C 180,E1 -5478.384,E2 -5478.384} C_VEL
LIN {X 0,Y 510.175,Z 819.855,A -85,B 0,C 180,E1 -5479.281,E2 -5479.281} C_VEL
LIN {X 0,Y 509.912,Z 829.107,A -85,B 0,C 180,E1 -5480.279,E2 -5480.279} C_VEL
LIN {X 0,Y 509.657,Z 838.117,A -85,B 0,C 180,E1 -5481.474,E2 -5481.474} C_VEL
LIN {X 0,Y 509.438,Z 845.37,A -85,B 0,C 180,E1 -5482.668,E2 -5482.668} C_VEL
LIN {X 0,Y 509.328,Z 850.266,A -85,B 0,C 180,E1 -5483.661,E2 -5483.661} C_VEL
LIN {X 0,Y 509.248,Z 855.025,A -85,B 0,C 180,E1 -5484.853,E2 -5484.853} C_VEL
LIN {X 0,Y 509.254,Z 858.664,A -85,B 0,C 180,E1 -5486.042,E2 -5486.042} C_VEL
LIN {X 0,Y 509.201,Z 860.538,A -85,B 0,C 180,E1 -5486.834,E2 -5486.834} C_VEL
LIN {X 0,Y 509.189,Z 861.944,A -85,B 0,C 180,E1 -5487.626,E2 -5487.626} C_VEL
LIN {X 0,Y 509.073,Z 863.554,A -85,B 0,C 180,E1 -5489.208,E2 -5489.208} C_VEL
LIN {X 0,Y 509.065,Z 863.771,A -85,B 0,C 180,E1 -5489.999,E2 -5489.999} C_VEL
LIN {X 0,Y 509.112,Z 862.944,A -85,B 0,C 180,E1 -5491.581,E2 -5491.581} C_VEL
LIN {X 0,Y 509.189,Z 861.945,A -85,B 0,C 180,E1 -5492.372,E2 -5492.372} C_VEL
LIN {X 0,Y 509.2,Z 860.537,A -85,B 0,C 180,E1 -5493.164,E2 -5493.164} C_VEL
LIN {X 0,Y 509.23,Z 857.577,A -85,B 0,C 180,E1 -5494.352,E2 -5494.352} C_VEL
LIN {X 0,Y 509.322,Z 853.572,A -85,B 0,C 180,E1 -5495.542,E2 -5495.542} C_VEL
LIN {X 0,Y 509.402,Z 847.862,A -85,B 0,C 180,E1 -5496.843,E2 -5496.843} C_VEL
LIN {X 0,Y 509.572,Z 840.667,A -85,B 0,C 180,E1 -5498.126,E2 -5498.126} C_VEL
LIN {X 0,Y 509.793,Z 832.305,A -85,B 0,C 180,E1 -5499.321,E2 -5499.321} C_VEL
LIN {X 0,Y 510.036,Z 823.726,A -85,B 0,C 180,E1 -5500.318,E2 -5500.318} C_VEL
LIN {X 0,Y 510.421,Z 813.136,A -85,B 0,C 180,E1 -5501.314,E2 -5501.314} C_VEL
LIN {X 0,Y 510.727,Z 802.027,A -85,B 0,C 180,E1 -5502.156,E2 -5502.156} C_VEL
LIN {X 0,Y 511.044,Z 791.143,A -85,B 0,C 180,E1 -5502.811,E2 -5502.811} C_VEL
LIN {X 0,Y 511.33,Z 779.267,A -85,B 0,C 180,E1 -5503.36,E2 -5503.36} C_VEL
LIN {X 0,Y 511.541,Z 766.484,A -85,B 0,C 180,E1 -5503.784,E2 -5503.784} C_VEL
LIN {X 0,Y 511.734,Z 753.346,A -85,B 0,C 180,E1 -5504.058,E2 -5504.058} C_VEL
LIN {X 0,Y 512.109,Z 661.633,A -85,B 0,C 180,E1 -5505.356,E2 -5505.356} C_VEL
LIN {X 0,Y 510.353,Z 650.04,A -85,B 0,C 180,E1 -5505.581,E2 -5505.581} C_VEL
LIN {X 0,Y 510.799,Z 630.623,A -85,B 0,C 180,E1 -5508.448,E2 -5508.448} C_VEL
LIN {X 0,Y 511.428,Z 609.683,A -85,B 0,C 180,E1 -5511.566,E2 -5511.566} C_VEL
LIN {X 0,Y 511.881,Z 592.913,A -85,B 0,C 180,E1 -5514.107,E2 -5514.107} C_VEL
LIN {X 0,Y 510.406,Z 584.458,A -85,B 0,C 180,E1 -5515.485,E2 -5515.485} C_VEL
LIN {X 0,Y 509.903,Z 581.972,A -85,B 0,C 180,E1 -5515.923,E2 -5515.923} C_VEL
LIN {X 0,Y 509.875,Z 581.975,A -85,B 0,C 180,E1 -5518.843,E2 -5518.843} C_VEL
LIN {X 0,Y 509.819,Z 581.979,A -85,B 0,C 180,E1 -5521.589,E2 -5521.589} C_VEL
LIN {X 0,Y 509.851,Z 581.979,A -85,B 0,C 180,E1 -5524.412,E2 -5524.412} C_VEL
LIN {X 0,Y 509.816,Z 581.977,A -85,B 0,C 180,E1 -5527.34,E2 -5527.34} C_VEL
LIN {X 0,Y 509.858,Z 581.979,A -85,B 0,C 180,E1 -5530.379,E2 -5530.379} C_VEL
LIN {X 0,Y 509.82,Z 581.979,A -85,B 0,C 180,E1 -5533.061,E2 -5533.061} C_VEL
LIN {X 0,Y 509.826,Z 581.977,A -85,B 0,C 180,E1 -5535.791,E2 -5535.791} C_VEL
LIN {X 0,Y 509.861,Z 581.977,A -85,B 0,C 180,E1 -5538.575,E2 -5538.575} C_VEL
LIN {X 0,Y 509.855,Z 581.971,A -85,B 0,C 180,E1 -5541.662,E2 -5541.662} C_VEL
LIN {X 0,Y 509.841,Z 581.978,A -85,B 0,C 180,E1 -5544.623,E2 -5544.623} C_VEL
LIN {X 0,Y 509.86,Z 581.97,A -85,B 0,C 180,E1 -5547.481,E2 -5547.481} C_VEL
LIN {X 0,Y 509.875,Z 581.974,A -85,B 0,C 180,E1 -5550.268,E2 -5550.268} C_VEL
LIN {X 0,Y 509.881,Z 581.968,A -85,B 0,C 180,E1 -5552.944,E2 -5552.944} C_VEL
LIN {X 0,Y 509.863,Z 581.969,A -85,B 0,C 180,E1 -5555.574,E2 -5555.574} C_VEL
LIN {X 0,Y 509.815,Z 581.98,A -85,B 0,C 180,E1 -5558.148,E2 -5558.148} C_VEL
LIN {X 0,Y 509.857,Z 581.975,A -85,B 0,C 180,E1 -5560.681,E2 -5560.681} C_VEL
LIN {X 0,Y 509.878,Z 581.968,A -85,B 0,C 180,E1 -5563.174,E2 -5563.174} C_VEL
LIN {X 0,Y 509.856,Z 581.97,A -85,B 0,C 180,E1 -5565.634,E2 -5565.634} C_VEL
LIN {X 0,Y 509.915,Z 581.966,A -85,B 0,C 180,E1 -5568.874,E2 -5568.874} C_VEL
LIN {X 0,Y 509.944,Z 581.965,A -85,B 0,C 180,E1 -5572.078,E2 -5572.078} C_VEL
LIN {X 0,Y 509.976,Z 581.962,A -85,B 0,C 180,E1 -5574.464,E2 -5574.464} C_VEL
LIN {X 0,Y 510.047,Z 581.948,A -85,B 0,C 180,E1 -5577.631,E2 -5577.631} C_VEL
LIN {X 0,Y 510.057,Z 581.949,A -85,B 0,C 180,E1 -5580.789,E2 -5580.789} C_VEL
LIN {X 0,Y 509.951,Z 581.96,A -85,B 0,C 180,E1 -5583.16,E2 -5583.16} C_VEL
LIN {X 0,Y 509.975,Z 581.965,A -85,B 0,C 180,E1 -5586.33,E2 -5586.33} C_VEL
LIN {X 0,Y 509.911,Z 581.968,A -85,B 0,C 180,E1 -5588.72,E2 -5588.72} C_VEL
LIN {X 0,Y 509.942,Z 581.965,A -85,B 0,C 180,E1 -5591.931,E2 -5591.931} C_VEL
LIN {X 0,Y 509.885,Z 581.974,A -85,B 0,C 180,E1 -5595.242,E2 -5595.242} C_VEL
LIN {X 0,Y 509.904,Z 581.98,A -85,B 0,C 180,E1 -5596.464,E2 -5596.464} C_VEL
LIN {X 0,Y 510.395,Z 587.125,A -85,B 0,C 180,E1 -5597.634,E2 -5597.634} C_VEL
LIN {X 0,Y 510.147,Z 595.591,A -85,B 0,C 180,E1 -5599.49,E2 -5599.49} C_VEL
LIN {X 0,Y 512.269,Z 606.383,A -85,B 0,C 180,E1 -5599.719,E2 -5599.719} C_VEL
LIN {X 0,Y 511.733,Z 701.999,A -85,B 0,C 180,E1 -5601.105,E2 -5601.105} C_VEL
LIN {X 0,Y 511.511,Z 715.102,A -85,B 0,C 180,E1 -5601.458,E2 -5601.458} C_VEL
LIN {X 0,Y 511.249,Z 727.429,A -85,B 0,C 180,E1 -5601.946,E2 -5601.946} C_VEL
LIN {X 0,Y 510.987,Z 738.571,A -85,B 0,C 180,E1 -5602.544,E2 -5602.544} C_VEL
LIN {X 0,Y 510.657,Z 749.961,A -85,B 0,C 180,E1 -5603.326,E2 -5603.326} C_VEL
LIN {X 0,Y 510.315,Z 760.002,A -85,B 0,C 180,E1 -5604.187,E2 -5604.187} C_VEL
LIN {X 0,Y 510.06,Z 768.676,A -85,B 0,C 180,E1 -5605.096,E2 -5605.096} C_VEL
LIN {X 0,Y 509.739,Z 777.157,A -85,B 0,C 180,E1 -5606.18,E2 -5606.18} C_VEL
LIN {X 0,Y 509.596,Z 784.254,A -85,B 0,C 180,E1 -5607.294,E2 -5607.294} C_VEL
LIN {X 0,Y 509.418,Z 791.113,A -85,B 0,C 180,E1 -5608.647,E2 -5608.647} C_VEL
LIN {X 0,Y 509.277,Z 795.651,A -85,B 0,C 180,E1 -5609.788,E2 -5609.788} C_VEL
LIN {X 0,Y 509.22,Z 799.781,A -85,B 0,C 180,E1 -5611.166,E2 -5611.166} C_VEL
LIN {X 0,Y 509.095,Z 802.748,A -85,B 0,C 180,E1 -5612.64,E2 -5612.64} C_VEL
LIN {X 0,Y 509.077,Z 804.248,A -85,B 0,C 180,E1 -5614.075,E2 -5614.075} C_VEL
LIN {X 0,Y 509.09,Z 804.395,A -85,B 0,C 180,E1 -5614.354,E2 -5614.354} C_VEL
LIN {X 0,Y 508.446,Z 804.618,A -85,B 0,C 180,E1 -5615.013,E2 -5615.013} C_VEL
LIN {X 0,Y 505.554,Z 804.411,A -85,B 0,C 180,E1 -5616.082,E2 -5616.082} C_VEL
LIN {X 0,Y 502.645,Z 803.552,A -85,B 0,C 180,E1 -5617.159,E2 -5617.159} C_VEL
LIN {X 0,Y 501.995,Z 802.508,A -85,B 0,C 180,E1 -5617.823,E2 -5617.823} C_VEL
LIN {X 0,Y 502.11,Z 799.998,A -85,B 0,C 180,E1 -5619.04,E2 -5619.04} C_VEL
LIN {X 0,Y 502.227,Z 795.565,A -85,B 0,C 180,E1 -5620.498,E2 -5620.498} C_VEL
LIN {X 0,Y 502.342,Z 789.826,A -85,B 0,C 180,E1 -5621.889,E2 -5621.889} C_VEL
LIN {X 0,Y 502.594,Z 782.517,A -85,B 0,C 180,E1 -5623.25,E2 -5623.25} C_VEL
LIN {X 0,Y 502.86,Z 773.734,A -85,B 0,C 180,E1 -5624.54,E2 -5624.54} C_VEL
LIN {X 0,Y 503.186,Z 765.006,A -85,B 0,C 180,E1 -5625.57,E2 -5625.57} C_VEL
LIN {X 0,Y 503.531,Z 754.95,A -85,B 0,C 180,E1 -5626.534,E2 -5626.534} C_VEL
LIN {X 0,Y 503.901,Z 743.198,A -85,B 0,C 180,E1 -5627.435,E2 -5627.435} C_VEL
LIN {X 0,Y 504.265,Z 731.26,A -85,B 0,C 180,E1 -5628.14,E2 -5628.14} C_VEL
LIN {X 0,Y 504.58,Z 718.35,A -85,B 0,C 180,E1 -5628.711,E2 -5628.711} C_VEL
LIN {X 0,Y 504.766,Z 706.241,A -85,B 0,C 180,E1 -5629.086,E2 -5629.086} C_VEL
LIN {X 0,Y 504.928,Z 691.127,A -85,B 0,C 180,E1 -5629.357,E2 -5629.357} C_VEL
LIN {X 0,Y 505.337,Z 606.643,A -85,B 0,C 180,E1 -5630.584,E2 -5630.584} C_VEL
LIN {X 0,Y 503.176,Z 595.46,A -85,B 0,C 180,E1 -5630.834,E2 -5630.834} C_VEL
LIN {X 0,Y 503.402,Z 586.834,A -85,B 0,C 180,E1 -5632.729,E2 -5632.729} C_VEL
LIN {X 0,Y 502.841,Z 582.853,A -85,B 0,C 180,E1 -5633.684,E2 -5633.684} C_VEL
LIN {X 0,Y 502.829,Z 582.846,A -85,B 0,C 180,E1 -5636.994,E2 -5636.994} C_VEL
LIN {X 0,Y 502.811,Z 582.856,A -85,B 0,C 180,E1 -5640.066,E2 -5640.066} C_VEL
LIN {X 0,Y 502.832,Z 582.847,A -85,B 0,C 180,E1 -5642.534,E2 -5642.534} C_VEL
LIN {X 0,Y 502.827,Z 582.845,A -85,B 0,C 180,E1 -5645.299,E2 -5645.299} C_VEL
LIN {X 0,Y 502.784,Z 582.855,A -85,B 0,C 180,E1 -5647.828,E2 -5647.828} C_VEL
LIN {X 0,Y 502.825,Z 582.851,A -85,B 0,C 180,E1 -5650.401,E2 -5650.401} C_VEL
LIN {X 0,Y 502.835,Z 582.845,A -85,B 0,C 180,E1 -5652.933,E2 -5652.933} C_VEL
LIN {X 0,Y 502.845,Z 582.843,A -85,B 0,C 180,E1 -5655.43,E2 -5655.43} C_VEL
LIN {X 0,Y 502.893,Z 582.841,A -85,B 0,C 180,E1 -5658.718,E2 -5658.718} C_VEL
LIN {X 0,Y 502.902,Z 582.839,A -85,B 0,C 180,E1 -5661.968,E2 -5661.968} C_VEL
LIN {X 0,Y 502.938,Z 582.84,A -85,B 0,C 180,E1 -5664.387,E2 -5664.387} C_VEL
LIN {X 0,Y 503.027,Z 582.82,A -85,B 0,C 180,E1 -5667.599,E2 -5667.599} C_VEL
LIN {X 0,Y 503.03,Z 582.822,A -85,B 0,C 180,E1 -5670.001,E2 -5670.001} C_VEL
LIN {X 0,Y 503.028,Z 582.826,A -85,B 0,C 180,E1 -5672.403,E2 -5672.403} C_VEL
LIN {X 0,Y 502.94,Z 582.831,A -85,B 0,C 180,E1 -5675.614,E2 -5675.614} C_VEL
LIN {X 0,Y 502.905,Z 582.836,A -85,B 0,C 180,E1 -5678.034,E2 -5678.034} C_VEL
LIN {X 0,Y 502.88,Z 582.84,A -85,B 0,C 180,E1 -5681.284,E2 -5681.284} C_VEL
LIN {X 0,Y 502.849,Z 582.848,A -85,B 0,C 180,E1 -5684.572,E2 -5684.572} C_VEL
LIN {X 0,Y 502.859,Z 582.841,A -85,B 0,C 180,E1 -5687.908,E2 -5687.908} C_VEL
LIN {X 0,Y 502.832,Z 582.848,A -85,B 0,C 180,E1 -5690.537,E2 -5690.537} C_VEL
LIN {X 0,Y 502.794,Z 582.857,A -85,B 0,C 180,E1 -5693.041,E2 -5693.041} C_VEL
LIN {X 0,Y 502.844,Z 582.844,A -85,B 0,C 180,E1 -5695.676,E2 -5695.676} C_VEL
LIN {X 0,Y 502.844,Z 582.844,A -85,B 0,C 180,E1 -5698.373,E2 -5698.373} C_VEL
LIN {X 0,Y 502.797,Z 582.853,A -85,B 0,C 180,E1 -5701.499,E2 -5701.499} C_VEL
LIN {X 0,Y 502.81,Z 582.847,A -85,B 0,C 180,E1 -5703.994,E2 -5703.994} C_VEL
LIN {X 0,Y 502.782,Z 582.86,A -85,B 0,C 180,E1 -5707.178,E2 -5707.178} C_VEL
LIN {X 0,Y 502.792,Z 582.85,A -85,B 0,C 180,E1 -5710.016,E2 -5710.016} C_VEL
LIN {X 0,Y 502.807,Z 582.848,A -85,B 0,C 180,E1 -5712.2,E2 -5712.2} C_VEL
LIN {X 0,Y 502.79,Z 582.858,A -85,B 0,C 180,E1 -5715.47,E2 -5715.47} C_VEL
LIN {X 0,Y 502.824,Z 582.848,A -85,B 0,C 180,E1 -5718.935,E2 -5718.935} C_VEL
LIN {X 0,Y 502.797,Z 582.851,A -85,B 0,C 180,E1 -5722.046,E2 -5722.046} C_VEL
LIN {X 0,Y 502.803,Z 582.85,A -85,B 0,C 180,E1 -5725.035,E2 -5725.035} C_VEL
LIN {X 0,Y 502.788,Z 582.855,A -85,B 0,C 180,E1 -5727.916,E2 -5727.916} C_VEL
LIN {X 0,Y 502.829,Z 582.845,A -85,B 0,C 180,E1 -5730.713,E2 -5730.713} C_VEL
LIN {X 0,Y 502.868,Z 582.845,A -85,B 0,C 180,E1 -5733.44,E2 -5733.44} C_VEL
LIN {X 0,Y 502.78,Z 582.855,A -85,B 0,C 180,E1 -5736.086,E2 -5736.086} C_VEL
LIN {X 0,Y 502.788,Z 582.85,A -85,B 0,C 180,E1 -5738.689,E2 -5738.689} C_VEL
LIN {X 0,Y 502.831,Z 582.846,A -85,B 0,C 180,E1 -5741.248,E2 -5741.248} C_VEL
LIN {X 0,Y 502.854,Z 582.843,A -85,B 0,C 180,E1 -5744.601,E2 -5744.601} C_VEL
LIN {X 0,Y 502.882,Z 582.847,A -85,B 0,C 180,E1 -5748.039,E2 -5748.039} C_VEL
LIN {X 0,Y 502.875,Z 582.839,A -85,B 0,C 180,E1 -5751.157,E2 -5751.157} C_VEL
LIN {X 0,Y 502.917,Z 582.836,A -85,B 0,C 180,E1 -5753.581,E2 -5753.581} C_VEL
LIN {X 0,Y 502.902,Z 582.837,A -85,B 0,C 180,E1 -5756.796,E2 -5756.796} C_VEL
LIN {X 0,Y 503.039,Z 582.819,A -85,B 0,C 180,E1 -5759.2,E2 -5759.2} C_VEL
LIN {X 0,Y 502.905,Z 582.837,A -85,B 0,C 180,E1 -5761.602,E2 -5761.602} C_VEL
LIN {X 0,Y 502.902,Z 582.836,A -85,B 0,C 180,E1 -5763.205,E2 -5763.205} C_VEL
LIN {X 0,Y 502.932,Z 582.84,A -85,B 0,C 180,E1 -5766.419,E2 -5766.419} C_VEL
LIN {X 0,Y 502.875,Z 582.841,A -85,B 0,C 180,E1 -5768.843,E2 -5768.843} C_VEL
LIN {X 0,Y 502.852,Z 582.847,A -85,B 0,C 180,E1 -5772.102,E2 -5772.102} C_VEL
LIN {X 0,Y 502.854,Z 582.842,A -85,B 0,C 180,E1 -5775.4,E2 -5775.4} C_VEL
LIN {X 0,Y 502.832,Z 582.85,A -85,B 0,C 180,E1 -5778.752,E2 -5778.752} C_VEL
LIN {X 0,Y 502.789,Z 582.85,A -85,B 0,C 180,E1 -5781.311,E2 -5781.311} C_VEL
LIN {X 0,Y 502.79,Z 582.85,A -85,B 0,C 180,E1 -5783.914,E2 -5783.914} C_VEL
LIN {X 0,Y 502.87,Z 582.847,A -85,B 0,C 180,E1 -5786.566,E2 -5786.566} C_VEL
LIN {X 0,Y 502.829,Z 582.846,A -85,B 0,C 180,E1 -5789.288,E2 -5789.288} C_VEL
LIN {X 0,Y 502.789,Z 582.851,A -85,B 0,C 180,E1 -5792.084,E2 -5792.084} C_VEL
LIN {X 0,Y 502.806,Z 582.855,A -85,B 0,C 180,E1 -5794.965,E2 -5794.965} C_VEL
LIN {X 0,Y 502.798,Z 582.849,A -85,B 0,C 180,E1 -5797.954,E2 -5797.954} C_VEL
LIN {X 0,Y 502.826,Z 582.853,A -85,B 0,C 180,E1 -5801.066,E2 -5801.066} C_VEL
LIN {X 0,Y 502.806,Z 582.85,A -85,B 0,C 180,E1 -5804.531,E2 -5804.531} C_VEL
LIN {X 0,Y 502.8,Z 582.849,A -85,B 0,C 180,E1 -5807.86,E2 -5807.86} C_VEL
LIN {X 0,Y 502.807,Z 582.855,A -85,B 0,C 180,E1 -5811.024,E2 -5811.024} C_VEL
LIN {X 0,Y 502.781,Z 582.851,A -85,B 0,C 180,E1 -5814.168,E2 -5814.168} C_VEL
LIN {X 0,Y 502.838,Z 582.851,A -85,B 0,C 180,E1 -5816.993,E2 -5816.993} C_VEL
LIN {X 0,Y 502.819,Z 582.849,A -85,B 0,C 180,E1 -5820.065,E2 -5820.065} C_VEL
LIN {X 0,Y 502.837,Z 582.848,A -85,B 0,C 180,E1 -5822.533,E2 -5822.533} C_VEL
LIN {X 0,Y 502.891,Z 582.997,A -85,B 0,C 180,E1 -5823.799,E2 -5823.799} C_VEL
LIN {X 0,Y 504.94,Z 593.27,A -85,B 0,C 180,E1 -5825.538,E2 -5825.538} C_VEL
LIN {X 0,Y 504.868,Z 600.944,A -85,B 0,C 180,E1 -5826.745,E2 -5826.745} C_VEL
LIN {X 0,Y 504.238,Z 619.651,A -85,B 0,C 180,E1 -5829.607,E2 -5829.607} C_VEL
LIN {X 0,Y 503.71,Z 638.996,A -85,B 0,C 180,E1 -5832.543,E2 -5832.543} C_VEL
LIN {X 0,Y 503.376,Z 649.944,A -85,B 0,C 180,E1 -5834.193,E2 -5834.193} C_VEL
LIN {X 0,Y 505.334,Z 663.628,A -85,B 0,C 180,E1 -5834.465,E2 -5834.465} C_VEL
LIN {X 0,Y 504.836,Z 758.631,A -85,B 0,C 180,E1 -5835.847,E2 -5835.847} C_VEL
LIN {X 0,Y 504.488,Z 771.918,A -85,B 0,C 180,E1 -5836.197,E2 -5836.197} C_VEL
LIN {X 0,Y 504.242,Z 784.686,A -85,B 0,C 180,E1 -5836.704,E2 -5836.704} C_VEL
LIN {X 0,Y 503.908,Z 796.603,A -85,B 0,C 180,E1 -5837.346,E2 -5837.346} C_VEL
LIN {X 0,Y 503.552,Z 807.769,A -85,B 0,C 180,E1 -5838.119,E2 -5838.119} C_VEL
LIN {X 0,Y 503.196,Z 818.319,A -85,B 0,C 180,E1 -5839.029,E2 -5839.029} C_VEL
LIN {X 0,Y 502.914,Z 826.947,A -85,B 0,C 180,E1 -5839.939,E2 -5839.939} C_VEL
LIN {X 0,Y 502.663,Z 834.906,A -85,B 0,C 180,E1 -5840.949,E2 -5840.949} C_VEL
LIN {X 0,Y 502.418,Z 842.682,A -85,B 0,C 180,E1 -5842.16,E2 -5842.16} C_VEL
LIN {X 0,Y 502.231,Z 849.457,A -85,B 0,C 180,E1 -5843.487,E2 -5843.487} C_VEL
LIN {X 0,Y 502.183,Z 854.607,A -85,B 0,C 180,E1 -5844.78,E2 -5844.78} C_VEL
LIN {X 0,Y 502.153,Z 858.249,A -85,B 0,C 180,E1 -5845.986,E2 -5845.986} C_VEL
LIN {X 0,Y 502.121,Z 860.127,A -85,B 0,C 180,E1 -5846.79,E2 -5846.79} C_VEL
LIN {X 0,Y 502.12,Z 861.536,A -85,B 0,C 180,E1 -5847.593,E2 -5847.593} C_VEL
LIN {X 0,Y 501.99,Z 863.145,A -85,B 0,C 180,E1 -5849.197,E2 -5849.197} C_VEL
LIN {X 0,Y 501.98,Z 863.36,A -85,B 0,C 180,E1 -5849.999,E2 -5849.999} C_VEL
LIN {X 0,Y 502.036,Z 862.528,A -85,B 0,C 180,E1 -5851.603,E2 -5851.603} C_VEL
LIN {X 0,Y 502.12,Z 861.527,A -85,B 0,C 180,E1 -5852.406,E2 -5852.406} C_VEL
LIN {X 0,Y 502.121,Z 860.111,A -85,B 0,C 180,E1 -5853.209,E2 -5853.209} C_VEL
LIN {X 0,Y 502.125,Z 857.141,A -85,B 0,C 180,E1 -5854.414,E2 -5854.414} C_VEL
LIN {X 0,Y 502.238,Z 853.126,A -85,B 0,C 180,E1 -5855.62,E2 -5855.62} C_VEL
LIN {X 0,Y 502.332,Z 847.045,A -85,B 0,C 180,E1 -5857.011,E2 -5857.011} C_VEL
LIN {X 0,Y 502.504,Z 840.191,A -85,B 0,C 180,E1 -5858.241,E2 -5858.241} C_VEL
LIN {X 0,Y 502.742,Z 831.808,A -85,B 0,C 180,E1 -5859.453,E2 -5859.453} C_VEL
LIN {X 0,Y 503.01,Z 823.207,A -85,B 0,C 180,E1 -5860.464,E2 -5860.464} C_VEL
LIN {X 0,Y 503.412,Z 812.591,A -85,B 0,C 180,E1 -5861.474,E2 -5861.474} C_VEL
LIN {X 0,Y 503.728,Z 801.451,A -85,B 0,C 180,E1 -5862.328,E2 -5862.328} C_VEL
LIN {X 0,Y 504.071,Z 790.527,A -85,B 0,C 180,E1 -5862.991,E2 -5862.991} C_VEL
LIN {X 0,Y 504.398,Z 778.583,A -85,B 0,C 180,E1 -5863.547,E2 -5863.547} C_VEL
LIN {X 0,Y 504.642,Z 765.713,A -85,B 0,C 180,E1 -5863.977,E2 -5863.977} C_VEL
LIN {X 0,Y 504.825,Z 752.349,A -85,B 0,C 180,E1 -5864.254,E2 -5864.254} C_VEL
LIN {X 0,Y 505.241,Z 662.443,A -85,B 0,C 180,E1 -5865.551,E2 -5865.551} C_VEL
LIN {X 0,Y 503.364,Z 649.393,A -85,B 0,C 180,E1 -5865.829,E2 -5865.829} C_VEL
LIN {X 0,Y 503.916,Z 628.75,A -85,B 0,C 180,E1 -5868.92,E2 -5868.92} C_VEL
LIN {X 0,Y 504.44,Z 610.613,A -85,B 0,C 180,E1 -5871.666,E2 -5871.666} C_VEL
LIN {X 0,Y 504.937,Z 593.906,A -85,B 0,C 180,E1 -5874.241,E2 -5874.241} C_VEL
LIN {X 0,Y 502.861,Z 582.849,A -85,B 0,C 180,E1 -5876.118,E2 -5876.118} C_VEL
LIN {X 0,Y 502.822,Z 582.85,A -85,B 0,C 180,E1 -5879.287,E2 -5879.287} C_VEL
LIN {X 0,Y 502.782,Z 582.858,A -85,B 0,C 180,E1 -5882.083,E2 -5882.083} C_VEL
LIN {X 0,Y 502.807,Z 582.853,A -85,B 0,C 180,E1 -5884.964,E2 -5884.964} C_VEL
LIN {X 0,Y 502.791,Z 582.854,A -85,B 0,C 180,E1 -5887.953,E2 -5887.953} C_VEL
LIN {X 0,Y 502.823,Z 582.851,A -85,B 0,C 180,E1 -5891.064,E2 -5891.064} C_VEL
LIN {X 0,Y 502.796,Z 582.858,A -85,B 0,C 180,E1 -5894.531,E2 -5894.531} C_VEL
LIN {X 0,Y 502.825,Z 582.849,A -85,B 0,C 180,E1 -5897.863,E2 -5897.863} C_VEL
LIN {X 0,Y 502.819,Z 582.849,A -85,B 0,C 180,E1 -5901.025,E2 -5901.025} C_VEL
LIN {X 0,Y 502.78,Z 582.855,A -85,B 0,C 180,E1 -5904.166,E2 -5904.166} C_VEL
LIN {X 0,Y 502.827,Z 582.848,A -85,B 0,C 180,E1 -5906.992,E2 -5906.992} C_VEL
LIN {X 0,Y 502.824,Z 582.849,A -85,B 0,C 180,E1 -5910.061,E2 -5910.061} C_VEL
LIN {X 0,Y 502.829,Z 582.852,A -85,B 0,C 180,E1 -5912.533,E2 -5912.533} C_VEL
LIN {X 0,Y 502.822,Z 582.846,A -85,B 0,C 180,E1 -5915.298,E2 -5915.298} C_VEL
LIN {X 0,Y 502.777,Z 582.853,A -85,B 0,C 180,E1 -5917.826,E2 -5917.826} C_VEL
LIN {X 0,Y 502.818,Z 582.854,A -85,B 0,C 180,E1 -5920.4,E2 -5920.4} C_VEL
LIN {X 0,Y 502.828,Z 582.848,A -85,B 0,C 180,E1 -5922.931,E2 -5922.931} C_VEL
LIN {X 0,Y 502.837,Z 582.844,A -85,B 0,C 180,E1 -5925.429,E2 -5925.429} C_VEL
LIN {X 0,Y 502.885,Z 582.843,A -85,B 0,C 180,E1 -5928.717,E2 -5928.717} C_VEL
LIN {X 0,Y 502.894,Z 582.842,A -85,B 0,C 180,E1 -5931.966,E2 -5931.966} C_VEL
LIN {X 0,Y 502.931,Z 582.84,A -85,B 0,C 180,E1 -5934.386,E2 -5934.386} C_VEL
LIN {X 0,Y 503.017,Z 582.824,A -85,B 0,C 180,E1 -5937.598,E2 -5937.598} C_VEL
LIN {X 0,Y 503.019,Z 582.827,A -85,B 0,C 180,E1 -5940,E2 -5940} C_VEL
LIN {X 0,Y 503.017,Z 582.831,A -85,B 0,C 180,E1 -5942.402,E2 -5942.402} C_VEL
LIN {X 0,Y 502.955,Z 582.833,A -85,B 0,C 180,E1 -5945.613,E2 -5945.613} C_VEL
LIN {X 0,Y 502.894,Z 582.845,A -85,B 0,C 180,E1 -5948.033,E2 -5948.033} C_VEL
LIN {X 0,Y 502.887,Z 582.84,A -85,B 0,C 180,E1 -5951.283,E2 -5951.283} C_VEL
LIN {X 0,Y 502.827,Z 582.856,A -85,B 0,C 180,E1 -5954.571,E2 -5954.571} C_VEL
LIN {X 0,Y 502.884,Z 583,A -85,B 0,C 180,E1 -5956.335,E2 -5956.335} C_VEL
LIN {X 0,Y 503.432,Z 587.906,A -85,B 0,C 180,E1 -5957.466,E2 -5957.466} C_VEL
LIN {X 0,Y 503.206,Z 596.044,A -85,B 0,C 180,E1 -5959.266,E2 -5959.266} C_VEL
LIN {X 0,Y 505.468,Z 607.61,A -85,B 0,C 180,E1 -5959.52,E2 -5959.52} C_VEL
LIN {X 0,Y 504.844,Z 701.891,A -85,B 0,C 180,E1 -5960.907,E2 -5960.907} C_VEL
LIN {X 0,Y 504.624,Z 714.926,A -85,B 0,C 180,E1 -5961.256,E2 -5961.256} C_VEL
LIN {X 0,Y 504.341,Z 727.984,A -85,B 0,C 180,E1 -5961.778,E2 -5961.778} C_VEL
LIN {X 0,Y 504.043,Z 739.971,A -85,B 0,C 180,E1 -5962.439,E2 -5962.439} C_VEL
LIN {X 0,Y 503.69,Z 750.944,A -85,B 0,C 180,E1 -5963.214,E2 -5963.214} C_VEL
LIN {X 0,Y 503.338,Z 761.076,A -85,B 0,C 180,E1 -5964.105,E2 -5964.105} C_VEL
LIN {X 0,Y 503.053,Z 769.409,A -85,B 0,C 180,E1 -5965,E2 -5965} C_VEL
LIN {X 0,Y 502.705,Z 778.048,A -85,B 0,C 180,E1 -5966.128,E2 -5966.128} C_VEL
LIN {X 0,Y 502.542,Z 785.052,A -85,B 0,C 180,E1 -5967.258,E2 -5967.258} C_VEL
LIN {X 0,Y 502.378,Z 791.828,A -85,B 0,C 180,E1 -5968.629,E2 -5968.629} C_VEL
LIN {X 0,Y 502.199,Z 796.405,A -85,B 0,C 180,E1 -5969.815,E2 -5969.815} C_VEL
LIN {X 0,Y 502.166,Z 800.385,A -85,B 0,C 180,E1 -5971.187,E2 -5971.187} C_VEL
LIN {X 0,Y 502.066,Z 802.375,A -85,B 0,C 180,E1 -5972.136,E2 -5972.136} C_VEL
LIN {X 0,Y 502.001,Z 803.821,A -85,B 0,C 180,E1 -5973.093,E2 -5973.093} C_VEL
LIN {X 0,Y 502.014,Z 804.813,A -85,B 0,C 180,E1 -5974.346,E2 -5974.346} C_VEL
LIN {X 0,Y 501.985,Z 804.837,A -85,B 0,C 180,E1 -5975.708,E2 -5975.708} C_VEL
LIN {X 0,Y 502.001,Z 803.709,A -85,B 0,C 180,E1 -5977.063,E2 -5977.063} C_VEL
LIN {X 0,Y 501.995,Z 802.508,A -85,B 0,C 180,E1 -5977.823,E2 -5977.823} C_VEL
LIN {X 0,Y 501.37,Z 801.353,A -85,B 0,C 180,E1 -5978.481,E2 -5978.481} C_VEL
LIN {X 0,Y 498.593,Z 798.956,A -85,B 0,C 180,E1 -5979.537,E2 -5979.537} C_VEL
LIN {X 0,Y 496.259,Z 796.559,A -85,B 0,C 180,E1 -5980.37,E2 -5980.37} C_VEL
LIN {X 0,Y 495.293,Z 794.375,A -85,B 0,C 180,E1 -5980.999,E2 -5980.999} C_VEL
LIN {X 0,Y 495.235,Z 793.556,A -85,B 0,C 180,E1 -5981.209,E2 -5981.209} C_VEL
LIN {X 0,Y 495.403,Z 786.889,A -85,B 0,C 180,E1 -5982.655,E2 -5982.655} C_VEL
LIN {X 0,Y 495.712,Z 778.843,A -85,B 0,C 180,E1 -5984.003,E2 -5984.003} C_VEL
LIN {X 0,Y 496.034,Z 770.671,A -85,B 0,C 180,E1 -5985.106,E2 -5985.106} C_VEL
LIN {X 0,Y 496.346,Z 761.985,A -85,B 0,C 180,E1 -5986.069,E2 -5986.069} C_VEL
LIN {X 0,Y 496.712,Z 751.511,A -85,B 0,C 180,E1 -5987.01,E2 -5987.01} C_VEL
LIN {X 0,Y 497.111,Z 739.841,A -85,B 0,C 180,E1 -5987.846,E2 -5987.846} C_VEL
LIN {X 0,Y 497.475,Z 728.409,A -85,B 0,C 180,E1 -5988.482,E2 -5988.482} C_VEL
LIN {X 0,Y 497.731,Z 715.473,A -85,B 0,C 180,E1 -5989.012,E2 -5989.012} C_VEL
LIN {X 0,Y 497.952,Z 702.26,A -85,B 0,C 180,E1 -5989.375,E2 -5989.375} C_VEL
LIN {X 0,Y 498.447,Z 607.164,A -85,B 0,C 180,E1 -5990.802,E2 -5990.802} C_VEL
LIN {X 0,Y 496.232,Z 595.799,A -85,B 0,C 180,E1 -5991.069,E2 -5991.069} C_VEL
LIN {X 0,Y 496.334,Z 587.049,A -85,B 0,C 180,E1 -5993.003,E2 -5993.003} C_VEL
LIN {X 0,Y 495.795,Z 583.731,A -85,B 0,C 180,E1 -5993.783,E2 -5993.783} C_VEL
LIN {X 0,Y 495.79,Z 583.724,A -85,B 0,C 180,E1 -5996.756,E2 -5996.756} C_VEL
LIN {X 0,Y 495.761,Z 583.733,A -85,B 0,C 180,E1 -5999.854,E2 -5999.854} C_VEL
LIN {X 0,Y 495.811,Z 583.719,A -85,B 0,C 180,E1 -6003.027,E2 -6003.027} C_VEL
LIN {X 0,Y 495.75,Z 583.73,A -85,B 0,C 180,E1 -6005.726,E2 -6005.726} C_VEL
LIN {X 0,Y 495.743,Z 583.733,A -85,B 0,C 180,E1 -6008.372,E2 -6008.372} C_VEL
LIN {X 0,Y 495.784,Z 583.723,A -85,B 0,C 180,E1 -6010.973,E2 -6010.973} C_VEL
LIN {X 0,Y 495.78,Z 583.724,A -85,B 0,C 180,E1 -6013.531,E2 -6013.531} C_VEL
LIN {X 0,Y 495.794,Z 583.727,A -85,B 0,C 180,E1 -6016.057,E2 -6016.057} C_VEL
LIN {X 0,Y 495.868,Z 583.718,A -85,B 0,C 180,E1 -6018.556,E2 -6018.556} C_VEL
LIN {X 0,Y 495.874,Z 583.713,A -85,B 0,C 180,E1 -6021.853,E2 -6021.853} C_VEL
LIN {X 0,Y 495.896,Z 583.716,A -85,B 0,C 180,E1 -6024.307,E2 -6024.307} C_VEL
LIN {X 0,Y 495.995,Z 583.696,A -85,B 0,C 180,E1 -6027.565,E2 -6027.565} C_VEL
LIN {X 0,Y 496.006,Z 583.7,A -85,B 0,C 180,E1 -6030.813,E2 -6030.813} C_VEL
LIN {X 0,Y 495.846,Z 583.716,A -85,B 0,C 180,E1 -6033.251,E2 -6033.251} C_VEL
LIN {X 0,Y 495.882,Z 583.717,A -85,B 0,C 180,E1 -6036.511,E2 -6036.511} C_VEL
LIN {X 0,Y 495.846,Z 583.72,A -85,B 0,C 180,E1 -6038.97,E2 -6038.97} C_VEL
LIN {X 0,Y 495.831,Z 583.717,A -85,B 0,C 180,E1 -6042.036,E2 -6042.036} C_VEL
LIN {X 0,Y 495.827,Z 583.718,A -85,B 0,C 180,E1 -6045.452,E2 -6045.452} C_VEL
LIN {X 0,Y 495.81,Z 583.72,A -85,B 0,C 180,E1 -6048.248,E2 -6048.248} C_VEL
LIN {X 0,Y 495.777,Z 583.73,A -85,B 0,C 180,E1 -6050.757,E2 -6050.757} C_VEL
LIN {X 0,Y 495.751,Z 583.73,A -85,B 0,C 180,E1 -6053.388,E2 -6053.388} C_VEL
LIN {X 0,Y 495.794,Z 583.721,A -85,B 0,C 180,E1 -6056.068,E2 -6056.068} C_VEL
LIN {X 0,Y 495.776,Z 583.729,A -85,B 0,C 180,E1 -6058.815,E2 -6058.815} C_VEL
LIN {X 0,Y 495.759,Z 583.727,A -85,B 0,C 180,E1 -6061.726,E2 -6061.726} C_VEL
LIN {X 0,Y 495.776,Z 583.726,A -85,B 0,C 180,E1 -6064.695,E2 -6064.695} C_VEL
LIN {X 0,Y 495.733,Z 583.733,A -85,B 0,C 180,E1 -6067.562,E2 -6067.562} C_VEL
LIN {X 0,Y 495.77,Z 583.726,A -85,B 0,C 180,E1 -6070.7,E2 -6070.7} C_VEL
LIN {X 0,Y 495.732,Z 583.73,A -85,B 0,C 180,E1 -6074.002,E2 -6074.002} C_VEL
LIN {X 0,Y 495.73,Z 583.734,A -85,B 0,C 180,E1 -6077.117,E2 -6077.117} C_VEL
LIN {X 0,Y 495.763,Z 583.727,A -85,B 0,C 180,E1 -6079.953,E2 -6079.953} C_VEL
LIN {X 0,Y 495.732,Z 583.729,A -85,B 0,C 180,E1 -6082.554,E2 -6082.554} C_VEL
LIN {X 0,Y 495.782,Z 583.73,A -85,B 0,C 180,E1 -6085.457,E2 -6085.457} C_VEL
LIN {X 0,Y 495.76,Z 583.726,A -85,B 0,C 180,E1 -6088.364,E2 -6088.364} C_VEL
LIN {X 0,Y 495.792,Z 583.728,A -85,B 0,C 180,E1 -6091.507,E2 -6091.507} C_VEL
LIN {X 0,Y 495.786,Z 583.728,A -85,B 0,C 180,E1 -6093.932,E2 -6093.932} C_VEL
LIN {X 0,Y 495.764,Z 583.726,A -85,B 0,C 180,E1 -6097.14,E2 -6097.14} C_VEL
LIN {X 0,Y 495.776,Z 583.728,A -85,B 0,C 180,E1 -6100.11,E2 -6100.11} C_VEL
LIN {X 0,Y 495.77,Z 583.724,A -85,B 0,C 180,E1 -6102.681,E2 -6102.681} C_VEL
LIN {X 0,Y 495.795,Z 583.722,A -85,B 0,C 180,E1 -6105.217,E2 -6105.217} C_VEL
LIN {X 0,Y 495.857,Z 583.715,A -85,B 0,C 180,E1 -6108.555,E2 -6108.555} C_VEL
LIN {X 0,Y 495.877,Z 583.717,A -85,B 0,C 180,E1 -6111.852,E2 -6111.852} C_VEL
LIN {X 0,Y 495.897,Z 583.714,A -85,B 0,C 180,E1 -6114.307,E2 -6114.307} C_VEL
LIN {X 0,Y 495.998,Z 583.697,A -85,B 0,C 180,E1 -6117.564,E2 -6117.564} C_VEL
LIN {X 0,Y 495.989,Z 583.698,A -85,B 0,C 180,E1 -6120.812,E2 -6120.812} C_VEL
LIN {X 0,Y 495.998,Z 583.702,A -85,B 0,C 180,E1 -6122.436,E2 -6122.436} C_VEL
LIN {X 0,Y 495.899,Z 583.71,A -85,B 0,C 180,E1 -6125.694,E2 -6125.694} C_VEL
LIN {X 0,Y 495.878,Z 583.717,A -85,B 0,C 180,E1 -6128.148,E2 -6128.148} C_VEL
LIN {X 0,Y 495.857,Z 583.713,A -85,B 0,C 180,E1 -6131.445,E2 -6131.445} C_VEL
LIN {X 0,Y 495.796,Z 583.725,A -85,B 0,C 180,E1 -6134.783,E2 -6134.783} C_VEL
LIN {X 0,Y 495.77,Z 583.724,A -85,B 0,C 180,E1 -6137.319,E2 -6137.319} C_VEL
LIN {X 0,Y 495.776,Z 583.724,A -85,B 0,C 180,E1 -6139.89,E2 -6139.89} C_VEL
LIN {X 0,Y 495.765,Z 583.73,A -85,B 0,C 180,E1 -6142.861,E2 -6142.861} C_VEL
LIN {X 0,Y 495.796,Z 583.722,A -85,B 0,C 180,E1 -6146.068,E2 -6146.068} C_VEL
LIN {X 0,Y 495.778,Z 583.731,A -85,B 0,C 180,E1 -6148.815,E2 -6148.815} C_VEL
LIN {X 0,Y 495.761,Z 583.725,A -85,B 0,C 180,E1 -6151.725,E2 -6151.725} C_VEL
LIN {X 0,Y 495.776,Z 583.731,A -85,B 0,C 180,E1 -6154.694,E2 -6154.694} C_VEL
LIN {X 0,Y 495.734,Z 583.729,A -85,B 0,C 180,E1 -6157.561,E2 -6157.561} C_VEL
LIN {X 0,Y 495.772,Z 583.73,A -85,B 0,C 180,E1 -6160.7,E2 -6160.7} C_VEL
LIN {X 0,Y 495.74,Z 583.728,A -85,B 0,C 180,E1 -6164.001,E2 -6164.001} C_VEL
LIN {X 0,Y 495.731,Z 583.737,A -85,B 0,C 180,E1 -6167.117,E2 -6167.117} C_VEL
LIN {X 0,Y 495.764,Z 583.725,A -85,B 0,C 180,E1 -6169.953,E2 -6169.953} C_VEL
LIN {X 0,Y 495.733,Z 583.73,A -85,B 0,C 180,E1 -6172.553,E2 -6172.553} C_VEL
LIN {X 0,Y 495.786,Z 583.729,A -85,B 0,C 180,E1 -6175.457,E2 -6175.457} C_VEL
LIN {X 0,Y 495.761,Z 583.727,A -85,B 0,C 180,E1 -6178.363,E2 -6178.363} C_VEL
LIN {X 0,Y 495.792,Z 583.73,A -85,B 0,C 180,E1 -6181.507,E2 -6181.507} C_VEL
LIN {X 0,Y 495.848,Z 583.772,A -85,B 0,C 180,E1 -6183.577,E2 -6183.577} C_VEL
LIN {X 0,Y 498.131,Z 595.751,A -85,B 0,C 180,E1 -6185.626,E2 -6185.626} C_VEL
LIN {X 0,Y 497.525,Z 613.755,A -85,B 0,C 180,E1 -6188.452,E2 -6188.452} C_VEL
LIN {X 0,Y 496.844,Z 633.54,A -85,B 0,C 180,E1 -6191.509,E2 -6191.509} C_VEL
LIN {X 0,Y 496.359,Z 649.562,A -85,B 0,C 180,E1 -6193.963,E2 -6193.963} C_VEL
LIN {X 0,Y 498.48,Z 664.186,A -85,B 0,C 180,E1 -6194.26,E2 -6194.26} C_VEL
LIN {X 0,Y 497.957,Z 757.895,A -85,B 0,C 180,E1 -6195.648,E2 -6195.648} C_VEL
LIN {X 0,Y 497.598,Z 771.304,A -85,B 0,C 180,E1 -6196.002,E2 -6196.002} C_VEL
LIN {X 0,Y 497.329,Z 784.124,A -85,B 0,C 180,E1 -6196.515,E2 -6196.515} C_VEL
LIN {X 0,Y 496.97,Z 795.129,A -85,B 0,C 180,E1 -6197.105,E2 -6197.105} C_VEL
LIN {X 0,Y 496.633,Z 805.977,A -85,B 0,C 180,E1 -6197.848,E2 -6197.848} C_VEL
LIN {X 0,Y 496.253,Z 816.767,A -85,B 0,C 180,E1 -6198.77,E2 -6198.77} C_VEL
LIN {X 0,Y 495.881,Z 826.486,A -85,B 0,C 180,E1 -6199.795,E2 -6199.795} C_VEL
LIN {X 0,Y 495.592,Z 834.457,A -85,B 0,C 180,E1 -6200.819,E2 -6200.819} C_VEL
LIN {X 0,Y 495.359,Z 842.248,A -85,B 0,C 180,E1 -6202.048,E2 -6202.048} C_VEL
LIN {X 0,Y 495.254,Z 847.579,A -85,B 0,C 180,E1 -6203.071,E2 -6203.071} C_VEL
LIN {X 0,Y 495.154,Z 852.747,A -85,B 0,C 180,E1 -6204.297,E2 -6204.297} C_VEL
LIN {X 0,Y 495.026,Z 856.753,A -85,B 0,C 180,E1 -6205.521,E2 -6205.521} C_VEL
LIN {X 0,Y 495.043,Z 859.715,A -85,B 0,C 180,E1 -6206.744,E2 -6206.744} C_VEL
LIN {X 0,Y 495.053,Z 861.127,A -85,B 0,C 180,E1 -6207.558,E2 -6207.558} C_VEL
LIN {X 0,Y 494.911,Z 862.734,A -85,B 0,C 180,E1 -6209.185,E2 -6209.185} C_VEL
LIN {X 0,Y 494.898,Z 862.948,A -85,B 0,C 180,E1 -6209.999,E2 -6209.999} C_VEL
LIN {X 0,Y 494.963,Z 862.113,A -85,B 0,C 180,E1 -6211.626,E2 -6211.626} C_VEL
LIN {X 0,Y 495.053,Z 861.107,A -85,B 0,C 180,E1 -6212.44,E2 -6212.44} C_VEL
LIN {X 0,Y 495.043,Z 859.686,A -85,B 0,C 180,E1 -6213.255,E2 -6213.255} C_VEL
LIN {X 0,Y 495.026,Z 856.705,A -85,B 0,C 180,E1 -6214.478,E2 -6214.478} C_VEL
LIN {X 0,Y 495.153,Z 852.68,A -85,B 0,C 180,E1 -6215.701,E2 -6215.701} C_VEL
LIN {X 0,Y 495.256,Z 846.482,A -85,B 0,C 180,E1 -6217.132,E2 -6217.132} C_VEL
LIN {X 0,Y 495.45,Z 839.715,A -85,B 0,C 180,E1 -6218.359,E2 -6218.359} C_VEL
LIN {X 0,Y 495.702,Z 831.312,A -85,B 0,C 180,E1 -6219.589,E2 -6219.589} C_VEL
LIN {X 0,Y 495.995,Z 822.687,A -85,B 0,C 180,E1 -6220.614,E2 -6220.614} C_VEL
LIN {X 0,Y 496.391,Z 812.044,A -85,B 0,C 180,E1 -6221.639,E2 -6221.639} C_VEL
LIN {X 0,Y 496.781,Z 800.389,A -85,B 0,C 180,E1 -6222.538,E2 -6222.538} C_VEL
LIN {X 0,Y 497.126,Z 787.911,A -85,B 0,C 180,E1 -6223.28,E2 -6223.28} C_VEL
LIN {X 0,Y 497.504,Z 775.283,A -85,B 0,C 180,E1 -6223.842,E2 -6223.842} C_VEL
LIN {X 0,Y 497.845,Z 763.095,A -85,B 0,C 180,E1 -6224.223,E2 -6224.223} C_VEL
LIN {X 0,Y 497.977,Z 749.556,A -85,B 0,C 180,E1 -6224.48,E2 -6224.48} C_VEL
LIN {X 0,Y 498.4,Z 663.188,A -85,B 0,C 180,E1 -6225.751,E2 -6225.751} C_VEL
LIN {X 0,Y 496.322,Z 648.925,A -85,B 0,C 180,E1 -6226.058,E2 -6226.058} C_VEL
LIN {X 0,Y 496.955,Z 628.269,A -85,B 0,C 180,E1 -6229.195,E2 -6229.195} C_VEL
LIN {X 0,Y 497.628,Z 607.42,A -85,B 0,C 180,E1 -6232.414,E2 -6232.414} C_VEL
LIN {X 0,Y 497.977,Z 594.903,A -85,B 0,C 180,E1 -6234.38,E2 -6234.38} C_VEL
LIN {X 0,Y 495.813,Z 583.727,A -85,B 0,C 180,E1 -6236.321,E2 -6236.321} C_VEL
LIN {X 0,Y 495.771,Z 583.733,A -85,B 0,C 180,E1 -6238.814,E2 -6238.814} C_VEL
LIN {X 0,Y 495.754,Z 583.732,A -85,B 0,C 180,E1 -6241.724,E2 -6241.724} C_VEL
LIN {X 0,Y 495.774,Z 583.732,A -85,B 0,C 180,E1 -6244.694,E2 -6244.694} C_VEL
LIN {X 0,Y 495.728,Z 583.732,A -85,B 0,C 180,E1 -6247.56,E2 -6247.56} C_VEL
LIN {X 0,Y 495.776,Z 583.732,A -85,B 0,C 180,E1 -6250.697,E2 -6250.697} C_VEL
LIN {X 0,Y 495.73,Z 583.735,A -85,B 0,C 180,E1 -6254,E2 -6254} C_VEL
LIN {X 0,Y 495.76,Z 583.729,A -85,B 0,C 180,E1 -6257.12,E2 -6257.12} C_VEL
LIN {X 0,Y 495.788,Z 583.731,A -85,B 0,C 180,E1 -6260.365,E2 -6260.365} C_VEL
LIN {X 0,Y 495.728,Z 583.729,A -85,B 0,C 180,E1 -6263.456,E2 -6263.456} C_VEL
LIN {X 0,Y 495.755,Z 583.733,A -85,B 0,C 180,E1 -6266.435,E2 -6266.435} C_VEL
LIN {X 0,Y 495.751,Z 583.727,A -85,B 0,C 180,E1 -6269.312,E2 -6269.312} C_VEL
LIN {X 0,Y 495.776,Z 583.726,A -85,B 0,C 180,E1 -6272.108,E2 -6272.108} C_VEL
LIN {X 0,Y 495.782,Z 583.727,A -85,B 0,C 180,E1 -6274.832,E2 -6274.832} C_VEL
LIN {X 0,Y 495.746,Z 583.727,A -85,B 0,C 180,E1 -6277.495,E2 -6277.495} C_VEL
LIN {X 0,Y 495.771,Z 583.728,A -85,B 0,C 180,E1 -6280.109,E2 -6280.109} C_VEL
LIN {X 0,Y 495.78,Z 583.729,A -85,B 0,C 180,E1 -6282.681,E2 -6282.681} C_VEL
LIN {X 0,Y 495.782,Z 583.723,A -85,B 0,C 180,E1 -6285.217,E2 -6285.217} C_VEL
LIN {X 0,Y 495.86,Z 583.721,A -85,B 0,C 180,E1 -6288.555,E2 -6288.555} C_VEL
LIN {X 0,Y 495.865,Z 583.716,A -85,B 0,C 180,E1 -6291.852,E2 -6291.852} C_VEL
LIN {X 0,Y 495.889,Z 583.718,A -85,B 0,C 180,E1 -6294.306,E2 -6294.306} C_VEL
LIN {X 0,Y 495.986,Z 583.699,A -85,B 0,C 180,E1 -6297.564,E2 -6297.564} C_VEL
LIN {X 0,Y 495.99,Z 583.703,A -85,B 0,C 180,E1 -6300,E2 -6300} C_VEL
LIN {X 0,Y 495.986,Z 583.707,A -85,B 0,C 180,E1 -6302.436,E2 -6302.436} C_VEL
LIN {X 0,Y 495.909,Z 583.712,A -85,B 0,C 180,E1 -6305.693,E2 -6305.693} C_VEL
LIN {X 0,Y 495.865,Z 583.722,A -85,B 0,C 180,E1 -6308.148,E2 -6308.148} C_VEL
LIN {X 0,Y 495.861,Z 583.715,A -85,B 0,C 180,E1 -6311.445,E2 -6311.445} C_VEL
LIN {X 0,Y 495.776,Z 583.735,A -85,B 0,C 180,E1 -6314.783,E2 -6314.783} C_VEL
LIN {X 0,Y 495.806,Z 583.81,A -85,B 0,C 180,E1 -6316.152,E2 -6316.152} C_VEL
LIN {X 0,Y 496.473,Z 588.68,A -85,B 0,C 180,E1 -6317.294,E2 -6317.294} C_VEL
LIN {X 0,Y 496.268,Z 596.512,A -85,B 0,C 180,E1 -6319.048,E2 -6319.048} C_VEL
LIN {X 0,Y 498.659,Z 608.285,A -85,B 0,C 180,E1 -6319.307,E2 -6319.307} C_VEL
LIN {X 0,Y 497.955,Z 702.529,A -85,B 0,C 180,E1 -6320.721,E2 -6320.721} C_VEL
LIN {X 0,Y 497.742,Z 716.239,A -85,B 0,C 180,E1 -6321.101,E2 -6321.101} C_VEL
LIN {X 0,Y 497.444,Z 728.527,A -85,B 0,C 180,E1 -6321.606,E2 -6321.606} C_VEL
LIN {X 0,Y 497.151,Z 739.626,A -85,B 0,C 180,E1 -6322.219,E2 -6322.219} C_VEL
LIN {X 0,Y 496.757,Z 751.115,A -85,B 0,C 180,E1 -6323.035,E2 -6323.035} C_VEL
LIN {X 0,Y 496.339,Z 762.163,A -85,B 0,C 180,E1 -6324.022,E2 -6324.022} C_VEL
LIN {X 0,Y 495.956,Z 772.211,A -85,B 0,C 180,E1 -6325.158,E2 -6325.158} C_VEL
LIN {X 0,Y 495.648,Z 780.939,A -85,B 0,C 180,E1 -6326.385,E2 -6326.385} C_VEL
LIN {X 0,Y 495.449,Z 788.255,A -85,B 0,C 180,E1 -6327.682,E2 -6327.682} C_VEL
LIN {X 0,Y 495.27,Z 793.513,A -85,B 0,C 180,E1 -6328.847,E2 -6328.847} C_VEL
LIN {X 0,Y 495.124,Z 798.687,A -85,B 0,C 180,E1 -6330.34,E2 -6330.34} C_VEL
LIN {X 0,Y 495.032,Z 802.024,A -85,B 0,C 180,E1 -6331.688,E2 -6331.688} C_VEL
LIN {X 0,Y 494.942,Z 804.272,A -85,B 0,C 180,E1 -6333.096,E2 -6333.096} C_VEL
LIN {X 0,Y 494.942,Z 805.312,A -85,B 0,C 180,E1 -6334.61,E2 -6334.61} C_VEL
LIN {X 0,Y 494.889,Z 805.112,A -85,B 0,C 180,E1 -6335.958,E2 -6335.958} C_VEL
LIN {X 0,Y 494.913,Z 803.368,A -85,B 0,C 180,E1 -6337.634,E2 -6337.634} C_VEL
LIN {X 0,Y 495.058,Z 800.182,A -85,B 0,C 180,E1 -6339.178,E2 -6339.178} C_VEL
LIN {X 0,Y 495.167,Z 796.812,A -85,B 0,C 180,E1 -6340.326,E2 -6340.326} C_VEL
LIN {X 0,Y 495.235,Z 793.556,A -85,B 0,C 180,E1 -6341.209,E2 -6341.209} C_VEL
LIN {X 0,Y 494.663,Z 791.064,A -85,B 0,C 180,E1 -6341.825,E2 -6341.825} C_VEL
LIN {X 0,Y 491.994,Z 786.608,A -85,B 0,C 180,E1 -6342.806,E2 -6342.806} C_VEL
LIN {X 0,Y 489.309,Z 781.538,A -85,B 0,C 180,E1 -6343.752,E2 -6343.752} C_VEL
LIN {X 0,Y 488.719,Z 778.016,A -85,B 0,C 180,E1 -6344.308,E2 -6344.308} C_VEL
LIN {X 0,Y 489.057,Z 770.324,A -85,B 0,C 180,E1 -6345.335,E2 -6345.335} C_VEL
LIN {X 0,Y 489.422,Z 760.242,A -85,B 0,C 180,E1 -6346.429,E2 -6346.429} C_VEL
LIN {X 0,Y 489.84,Z 749.974,A -85,B 0,C 180,E1 -6347.329,E2 -6347.329} C_VEL
LIN {X 0,Y 490.237,Z 738.832,A -85,B 0,C 180,E1 -6348.111,E2 -6348.111} C_VEL
LIN {X 0,Y 490.638,Z 726.238,A -85,B 0,C 180,E1 -6348.785,E2 -6348.785} C_VEL
LIN {X 0,Y 490.91,Z 713.114,A -85,B 0,C 180,E1 -6349.297,E2 -6349.297} C_VEL
LIN {X 0,Y 491.13,Z 699.803,A -85,B 0,C 180,E1 -6349.625,E2 -6349.625} C_VEL
LIN {X 0,Y 491.741,Z 608.759,A -85,B 0,C 180,E1 -6351.003,E2 -6351.003} C_VEL
LIN {X 0,Y 489.259,Z 596.174,A -85,B 0,C 180,E1 -6351.297,E2 -6351.297} C_VEL
LIN {X 0,Y 489.429,Z 588.941,A -85,B 0,C 180,E1 -6352.909,E2 -6352.909} C_VEL
LIN {X 0,Y 488.744,Z 584.608,A -85,B 0,C 180,E1 -6353.939,E2 -6353.939} C_VEL
LIN {X 0,Y 488.735,Z 584.602,A -85,B 0,C 180,E1 -6356.878,E2 -6356.878} C_VEL
LIN {X 0,Y 488.72,Z 584.609,A -85,B 0,C 180,E1 -6359.782,E2 -6359.782} C_VEL
LIN {X 0,Y 488.789,Z 584.594,A -85,B 0,C 180,E1 -6363.057,E2 -6363.057} C_VEL
LIN {X 0,Y 488.693,Z 584.613,A -85,B 0,C 180,E1 -6366.256,E2 -6366.256} C_VEL
LIN {X 0,Y 488.744,Z 584.599,A -85,B 0,C 180,E1 -6369.177,E2 -6369.177} C_VEL
LIN {X 0,Y 488.758,Z 584.599,A -85,B 0,C 180,E1 -6371.629,E2 -6371.629} C_VEL
LIN {X 0,Y 488.762,Z 584.598,A -85,B 0,C 180,E1 -6375.001,E2 -6375.001} C_VEL
LIN {X 0,Y 488.83,Z 584.597,A -85,B 0,C 180,E1 -6378.389,E2 -6378.389} C_VEL
LIN {X 0,Y 488.818,Z 584.591,A -85,B 0,C 180,E1 -6381.735,E2 -6381.735} C_VEL
LIN {X 0,Y 488.855,Z 584.591,A -85,B 0,C 180,E1 -6384.225,E2 -6384.225} C_VEL
LIN {X 0,Y 488.963,Z 584.572,A -85,B 0,C 180,E1 -6387.53,E2 -6387.53} C_VEL
LIN {X 0,Y 488.956,Z 584.578,A -85,B 0,C 180,E1 -6390.824,E2 -6390.824} C_VEL
LIN {X 0,Y 488.964,Z 584.579,A -85,B 0,C 180,E1 -6392.472,E2 -6392.472} C_VEL
LIN {X 0,Y 488.857,Z 584.585,A -85,B 0,C 180,E1 -6395.777,E2 -6395.777} C_VEL
LIN {X 0,Y 488.821,Z 584.593,A -85,B 0,C 180,E1 -6398.267,E2 -6398.267} C_VEL
LIN {X 0,Y 488.809,Z 584.591,A -85,B 0,C 180,E1 -6401.613,E2 -6401.613} C_VEL
LIN {X 0,Y 488.765,Z 584.603,A -85,B 0,C 180,E1 -6405.001,E2 -6405.001} C_VEL
LIN {X 0,Y 488.758,Z 584.601,A -85,B 0,C 180,E1 -6408.443,E2 -6408.443} C_VEL
LIN {X 0,Y 488.71,Z 584.611,A -85,B 0,C 180,E1 -6411.071,E2 -6411.071} C_VEL
LIN {X 0,Y 488.692,Z 584.606,A -85,B 0,C 180,E1 -6413.746,E2 -6413.746} C_VEL
LIN {X 0,Y 488.796,Z 584.601,A -85,B 0,C 180,E1 -6416.944,E2 -6416.944} C_VEL
LIN {X 0,Y 488.713,Z 584.604,A -85,B 0,C 180,E1 -6420.363,E2 -6420.363} C_VEL
LIN {X 0,Y 488.739,Z 584.604,A -85,B 0,C 180,E1 -6423.485,E2 -6423.485} C_VEL
LIN {X 0,Y 488.687,Z 584.607,A -85,B 0,C 180,E1 -6426.355,E2 -6426.355} C_VEL
LIN {X 0,Y 488.706,Z 584.614,A -85,B 0,C 180,E1 -6429.255,E2 -6429.255} C_VEL
LIN {X 0,Y 488.711,Z 584.608,A -85,B 0,C 180,E1 -6431.6,E2 -6431.6} C_VEL
LIN {X 0,Y 488.705,Z 584.606,A -85,B 0,C 180,E1 -6434.803,E2 -6434.803} C_VEL
LIN {X 0,Y 488.696,Z 584.614,A -85,B 0,C 180,E1 -6437.475,E2 -6437.475} C_VEL
LIN {X 0,Y 488.737,Z 584.606,A -85,B 0,C 180,E1 -6439.677,E2 -6439.677} C_VEL
LIN {X 0,Y 488.683,Z 584.608,A -85,B 0,C 180,E1 -6442.841,E2 -6442.841} C_VEL
LIN {X 0,Y 488.735,Z 584.605,A -85,B 0,C 180,E1 -6445.888,E2 -6445.888} C_VEL
LIN {X 0,Y 488.696,Z 584.606,A -85,B 0,C 180,E1 -6448.821,E2 -6448.821} C_VEL
LIN {X 0,Y 488.749,Z 584.608,A -85,B 0,C 180,E1 -6451.672,E2 -6451.672} C_VEL
LIN {X 0,Y 488.732,Z 584.602,A -85,B 0,C 180,E1 -6454.443,E2 -6454.443} C_VEL
LIN {X 0,Y 488.726,Z 584.603,A -85,B 0,C 180,E1 -6457.153,E2 -6457.153} C_VEL
LIN {X 0,Y 488.73,Z 584.611,A -85,B 0,C 180,E1 -6459.811,E2 -6459.811} C_VEL
LIN {X 0,Y 488.72,Z 584.604,A -85,B 0,C 180,E1 -6462.423,E2 -6462.423} C_VEL
LIN {X 0,Y 488.767,Z 584.596,A -85,B 0,C 180,E1 -6465,E2 -6465} C_VEL
LIN {X 0,Y 488.811,Z 584.594,A -85,B 0,C 180,E1 -6468.388,E2 -6468.388} C_VEL
LIN {X 0,Y 488.821,Z 584.594,A -85,B 0,C 180,E1 -6471.734,E2 -6471.734} C_VEL
LIN {X 0,Y 488.855,Z 584.593,A -85,B 0,C 180,E1 -6474.224,E2 -6474.224} C_VEL
LIN {X 0,Y 488.966,Z 584.573,A -85,B 0,C 180,E1 -6477.529,E2 -6477.529} C_VEL
LIN {X 0,Y 488.94,Z 584.576,A -85,B 0,C 180,E1 -6480.824,E2 -6480.824} C_VEL
LIN {X 0,Y 488.966,Z 584.577,A -85,B 0,C 180,E1 -6482.471,E2 -6482.471} C_VEL
LIN {X 0,Y 488.859,Z 584.587,A -85,B 0,C 180,E1 -6485.776,E2 -6485.776} C_VEL
LIN {X 0,Y 488.822,Z 584.598,A -85,B 0,C 180,E1 -6488.266,E2 -6488.266} C_VEL
LIN {X 0,Y 488.811,Z 584.591,A -85,B 0,C 180,E1 -6491.612,E2 -6491.612} C_VEL
LIN {X 0,Y 488.768,Z 584.598,A -85,B 0,C 180,E1 -6495,E2 -6495} C_VEL
LIN {X 0,Y 488.753,Z 584.606,A -85,B 0,C 180,E1 -6498.442,E2 -6498.442} C_VEL
LIN {X 0,Y 488.712,Z 584.606,A -85,B 0,C 180,E1 -6501.071,E2 -6501.071} C_VEL
LIN {X 0,Y 488.694,Z 584.606,A -85,B 0,C 180,E1 -6503.746,E2 -6503.746} C_VEL
LIN {X 0,Y 488.797,Z 584.598,A -85,B 0,C 180,E1 -6506.943,E2 -6506.943} C_VEL
LIN {X 0,Y 488.715,Z 584.607,A -85,B 0,C 180,E1 -6510.363,E2 -6510.363} C_VEL
LIN {X 0,Y 488.74,Z 584.601,A -85,B 0,C 180,E1 -6513.484,E2 -6513.484} C_VEL
LIN {X 0,Y 488.688,Z 584.609,A -85,B 0,C 180,E1 -6516.354,E2 -6516.354} C_VEL
LIN {X 0,Y 488.707,Z 584.608,A -85,B 0,C 180,E1 -6519.254,E2 -6519.254} C_VEL
LIN {X 0,Y 488.713,Z 584.604,A -85,B 0,C 180,E1 -6521.6,E2 -6521.6} C_VEL
LIN {X 0,Y 488.718,Z 584.609,A -85,B 0,C 180,E1 -6524.801,E2 -6524.801} C_VEL
LIN {X 0,Y 488.697,Z 584.608,A -85,B 0,C 180,E1 -6527.474,E2 -6527.474} C_VEL
LIN {X 0,Y 488.738,Z 584.602,A -85,B 0,C 180,E1 -6529.676,E2 -6529.676} C_VEL
LIN {X 0,Y 488.685,Z 584.611,A -85,B 0,C 180,E1 -6532.841,E2 -6532.841} C_VEL
LIN {X 0,Y 488.738,Z 584.603,A -85,B 0,C 180,E1 -6535.887,E2 -6535.887} C_VEL
LIN {X 0,Y 488.697,Z 584.61,A -85,B 0,C 180,E1 -6538.82,E2 -6538.82} C_VEL
LIN {X 0,Y 488.749,Z 584.606,A -85,B 0,C 180,E1 -6541.671,E2 -6541.671} C_VEL
LIN {X 0,Y 488.809,Z 584.717,A -85,B 0,C 180,E1 -6543.378,E2 -6543.378} C_VEL
LIN {X 0,Y 491.16,Z 596.791,A -85,B 0,C 180,E1 -6545.482,E2 -6545.482} C_VEL
LIN {X 0,Y 490.806,Z 609.236,A -85,B 0,C 180,E1 -6547.477,E2 -6547.477} C_VEL
LIN {X 0,Y 490.036,Z 629.961,A -85,B 0,C 180,E1 -6550.739,E2 -6550.739} C_VEL
LIN {X 0,Y 489.388,Z 649.324,A -85,B 0,C 180,E1 -6553.736,E2 -6553.736} C_VEL
LIN {X 0,Y 491.629,Z 665.671,A -85,B 0,C 180,E1 -6554.063,E2 -6554.063} C_VEL
LIN {X 0,Y 491.03,Z 758.339,A -85,B 0,C 180,E1 -6555.467,E2 -6555.467} C_VEL
LIN {X 0,Y 490.648,Z 772.205,A -85,B 0,C 180,E1 -6555.853,E2 -6555.853} C_VEL
LIN {X 0,Y 490.377,Z 784.676,A -85,B 0,C 180,E1 -6556.373,E2 -6556.373} C_VEL
LIN {X 0,Y 489.948,Z 796.566,A -85,B 0,C 180,E1 -6557.045,E2 -6557.045} C_VEL
LIN {X 0,Y 489.535,Z 808.085,A -85,B 0,C 180,E1 -6557.879,E2 -6557.879} C_VEL
LIN {X 0,Y 489.14,Z 818.442,A -85,B 0,C 180,E1 -6558.815,E2 -6558.815} C_VEL
LIN {X 0,Y 488.781,Z 827.742,A -85,B 0,C 180,E1 -6559.854,E2 -6559.854} C_VEL
LIN {X 0,Y 488.451,Z 836.786,A -85,B 0,C 180,E1 -6561.101,E2 -6561.101} C_VEL
LIN {X 0,Y 488.221,Z 844.072,A -85,B 0,C 180,E1 -6562.347,E2 -6562.347} C_VEL
LIN {X 0,Y 488.037,Z 849.657,A -85,B 0,C 180,E1 -6563.536,E2 -6563.536} C_VEL
LIN {X 0,Y 488.052,Z 853.771,A -85,B 0,C 180,E1 -6564.628,E2 -6564.628} C_VEL
LIN {X 0,Y 487.951,Z 857.419,A -85,B 0,C 180,E1 -6565.869,E2 -6565.869} C_VEL
LIN {X 0,Y 487.967,Z 859.304,A -85,B 0,C 180,E1 -6566.696,E2 -6566.696} C_VEL
LIN {X 0,Y 487.959,Z 860.716,A -85,B 0,C 180,E1 -6567.523,E2 -6567.523} C_VEL
LIN {X 0,Y 487.893,Z 861.718,A -85,B 0,C 180,E1 -6568.348,E2 -6568.348} C_VEL
LIN {X 0,Y 487.819,Z 862.537,A -85,B 0,C 180,E1 -6569.999,E2 -6569.999} C_VEL
LIN {X 0,Y 487.893,Z 861.698,A -85,B 0,C 180,E1 -6571.65,E2 -6571.65} C_VEL
LIN {X 0,Y 487.972,Z 860.685,A -85,B 0,C 180,E1 -6572.475,E2 -6572.475} C_VEL
LIN {X 0,Y 487.967,Z 859.26,A -85,B 0,C 180,E1 -6573.302,E2 -6573.302} C_VEL
LIN {X 0,Y 487.936,Z 856.27,A -85,B 0,C 180,E1 -6574.543,E2 -6574.543} C_VEL
LIN {X 0,Y 488.049,Z 852.233,A -85,B 0,C 180,E1 -6575.784,E2 -6575.784} C_VEL
LIN {X 0,Y 488.182,Z 846.021,A -85,B 0,C 180,E1 -6577.236,E2 -6577.236} C_VEL
LIN {X 0,Y 488.378,Z 839.235,A -85,B 0,C 180,E1 -6578.481,E2 -6578.481} C_VEL
LIN {X 0,Y 488.636,Z 830.814,A -85,B 0,C 180,E1 -6579.729,E2 -6579.729} C_VEL
LIN {X 0,Y 488.958,Z 822.164,A -85,B 0,C 180,E1 -6580.768,E2 -6580.768} C_VEL
LIN {X 0,Y 489.331,Z 811.492,A -85,B 0,C 180,E1 -6581.809,E2 -6581.809} C_VEL
LIN {X 0,Y 489.736,Z 801.215,A -85,B 0,C 180,E1 -6582.619,E2 -6582.619} C_VEL
LIN {X 0,Y 490.129,Z 789.283,A -85,B 0,C 180,E1 -6583.368,E2 -6583.368} C_VEL
LIN {X 0,Y 490.538,Z 777.214,A -85,B 0,C 180,E1 -6583.937,E2 -6583.937} C_VEL
LIN {X 0,Y 490.858,Z 765.091,A -85,B 0,C 180,E1 -6584.351,E2 -6584.351} C_VEL
LIN {X 0,Y 491.051,Z 751.971,A -85,B 0,C 180,E1 -6584.636,E2 -6584.636} C_VEL
LIN {X 0,Y 491.568,Z 664.152,A -85,B 0,C 180,E1 -6585.954,E2 -6585.954} C_VEL
LIN {X 0,Y 489.349,Z 648.569,A -85,B 0,C 180,E1 -6586.274,E2 -6586.274} C_VEL
LIN {X 0,Y 489.991,Z 627.833,A -85,B 0,C 180,E1 -6589.479,E2 -6589.479} C_VEL
LIN {X 0,Y 490.68,Z 608.398,A -85,B 0,C 180,E1 -6592.527,E2 -6592.527} C_VEL
LIN {X 0,Y 491.002,Z 595.918,A -85,B 0,C 180,E1 -6594.524,E2 -6594.524} C_VEL
LIN {X 0,Y 488.805,Z 584.601,A -85,B 0,C 180,E1 -6596.506,E2 -6596.506} C_VEL
LIN {X 0,Y 488.722,Z 584.607,A -85,B 0,C 180,E1 -6599.269,E2 -6599.269} C_VEL
LIN {X 0,Y 488.701,Z 584.613,A -85,B 0,C 180,E1 -6602.146,E2 -6602.146} C_VEL
LIN {X 0,Y 488.72,Z 584.607,A -85,B 0,C 180,E1 -6605.113,E2 -6605.113} C_VEL
LIN {X 0,Y 488.68,Z 584.614,A -85,B 0,C 180,E1 -6608.199,E2 -6608.199} C_VEL
LIN {X 0,Y 488.745,Z 584.609,A -85,B 0,C 180,E1 -6610.348,E2 -6610.348} C_VEL
LIN {X 0,Y 488.682,Z 584.611,A -85,B 0,C 180,E1 -6613.653,E2 -6613.653} C_VEL
LIN {X 0,Y 488.712,Z 584.613,A -85,B 0,C 180,E1 -6616.348,E2 -6616.348} C_VEL
LIN {X 0,Y 488.731,Z 584.603,A -85,B 0,C 180,E1 -6619.676,E2 -6619.676} C_VEL
LIN {X 0,Y 488.678,Z 584.615,A -85,B 0,C 180,E1 -6622.276,E2 -6622.276} C_VEL
LIN {X 0,Y 488.723,Z 584.604,A -85,B 0,C 180,E1 -6625.051,E2 -6625.051} C_VEL
LIN {X 0,Y 488.7,Z 584.609,A -85,B 0,C 180,E1 -6628.044,E2 -6628.044} C_VEL
LIN {X 0,Y 488.727,Z 584.604,A -85,B 0,C 180,E1 -6630.73,E2 -6630.73} C_VEL
LIN {X 0,Y 488.759,Z 584.597,A -85,B 0,C 180,E1 -6633.528,E2 -6633.528} C_VEL
LIN {X 0,Y 488.687,Z 584.614,A -85,B 0,C 180,E1 -6636.254,E2 -6636.254} C_VEL
LIN {X 0,Y 488.738,Z 584.6,A -85,B 0,C 180,E1 -6639.175,E2 -6639.175} C_VEL
LIN {X 0,Y 488.751,Z 584.601,A -85,B 0,C 180,E1 -6641.627,E2 -6641.627} C_VEL
LIN {X 0,Y 488.754,Z 584.599,A -85,B 0,C 180,E1 -6644.999,E2 -6644.999} C_VEL
LIN {X 0,Y 488.821,Z 584.598,A -85,B 0,C 180,E1 -6648.388,E2 -6648.388} C_VEL
LIN {X 0,Y 488.81,Z 584.594,A -85,B 0,C 180,E1 -6651.733,E2 -6651.733} C_VEL
LIN {X 0,Y 488.848,Z 584.595,A -85,B 0,C 180,E1 -6654.224,E2 -6654.224} C_VEL
LIN {X 0,Y 488.954,Z 584.575,A -85,B 0,C 180,E1 -6657.528,E2 -6657.528} C_VEL
LIN {X 0,Y 488.961,Z 584.579,A -85,B 0,C 180,E1 -6660,E2 -6660} C_VEL
LIN {X 0,Y 488.954,Z 584.582,A -85,B 0,C 180,E1 -6662.471,E2 -6662.471} C_VEL
LIN {X 0,Y 488.865,Z 584.59,A -85,B 0,C 180,E1 -6665.776,E2 -6665.776} C_VEL
LIN {X 0,Y 488.81,Z 584.601,A -85,B 0,C 180,E1 -6668.266,E2 -6668.266} C_VEL
LIN {X 0,Y 488.822,Z 584.593,A -85,B 0,C 180,E1 -6671.612,E2 -6671.612} C_VEL
LIN {X 0,Y 488.788,Z 584.605,A -85,B 0,C 180,E1 -6675.564,E2 -6675.564} C_VEL
LIN {X 0,Y 488.784,Z 584.65,A -85,B 0,C 180,E1 -6675.961,E2 -6675.961} C_VEL
LIN {X 0,Y 489.502,Z 589.499,A -85,B 0,C 180,E1 -6677.117,E2 -6677.117} C_VEL
LIN {X 0,Y 489.336,Z 596.924,A -85,B 0,C 180,E1 -6678.802,E2 -6678.802} C_VEL
LIN {X 0,Y 491.853,Z 609.701,A -85,B 0,C 180,E1 -6679.102,E2 -6679.102} C_VEL
LIN {X 0,Y 491.074,Z 702.988,A -85,B 0,C 180,E1 -6680.526,E2 -6680.526} C_VEL
LIN {X 0,Y 490.85,Z 716.131,A -85,B 0,C 180,E1 -6680.892,E2 -6680.892} C_VEL
LIN {X 0,Y 490.542,Z 728.798,A -85,B 0,C 180,E1 -6681.415,E2 -6681.415} C_VEL
LIN {X 0,Y 490.287,Z 739.229,A -85,B 0,C 180,E1 -6681.993,E2 -6681.993} C_VEL
LIN {X 0,Y 489.859,Z 750.548,A -85,B 0,C 180,E1 -6682.791,E2 -6682.791} C_VEL
LIN {X 0,Y 489.447,Z 760.903,A -85,B 0,C 180,E1 -6683.707,E2 -6683.707} C_VEL
LIN {X 0,Y 489.087,Z 769.429,A -85,B 0,C 180,E1 -6684.628,E2 -6684.628} C_VEL
LIN {X 0,Y 488.733,Z 778.232,A -85,B 0,C 180,E1 -6685.785,E2 -6685.785} C_VEL
LIN {X 0,Y 488.465,Z 786.242,A -85,B 0,C 180,E1 -6687.111,E2 -6687.111} C_VEL
LIN {X 0,Y 488.285,Z 792.251,A -85,B 0,C 180,E1 -6688.358,E2 -6688.358} C_VEL
LIN {X 0,Y 488.074,Z 797.58,A -85,B 0,C 180,E1 -6689.772,E2 -6689.772} C_VEL
LIN {X 0,Y 487.998,Z 801.561,A -85,B 0,C 180,E1 -6691.229,E2 -6691.229} C_VEL
LIN {X 0,Y 487.913,Z 803.463,A -85,B 0,C 180,E1 -6692.205,E2 -6692.205} C_VEL
LIN {X 0,Y 487.841,Z 804.939,A -85,B 0,C 180,E1 -6693.327,E2 -6693.327} C_VEL
LIN {X 0,Y 487.839,Z 805.76,A -85,B 0,C 180,E1 -6694.801,E2 -6694.801} C_VEL
LIN {X 0,Y 487.819,Z 805.373,A -85,B 0,C 180,E1 -6696.219,E2 -6696.219} C_VEL
LIN {X 0,Y 487.834,Z 803.878,A -85,B 0,C 180,E1 -6697.595,E2 -6697.595} C_VEL
LIN {X 0,Y 487.949,Z 801.305,A -85,B 0,C 180,E1 -6698.945,E2 -6698.945} C_VEL
LIN {X 0,Y 488.105,Z 797.247,A -85,B 0,C 180,E1 -6700.386,E2 -6700.386} C_VEL
LIN {X 0,Y 488.198,Z 792.086,A -85,B 0,C 180,E1 -6701.744,E2 -6701.744} C_VEL
LIN {X 0,Y 488.433,Z 786.223,A -85,B 0,C 180,E1 -6702.955,E2 -6702.955} C_VEL
LIN {X 0,Y 488.708,Z 779.004,A -85,B 0,C 180,E1 -6704.161,E2 -6704.161} C_VEL
LIN {X 0,Y 488.719,Z 778.016,A -85,B 0,C 180,E1 -6704.308,E2 -6704.308} C_VEL
LIN {X 0,Y 488.15,Z 774.338,A -85,B 0,C 180,E1 -6704.849,E2 -6704.849} C_VEL
LIN {X 0,Y 485.581,Z 768.095,A -85,B 0,C 180,E1 -6705.707,E2 -6705.707} C_VEL
LIN {X 0,Y 483.097,Z 761.302,A -85,B 0,C 180,E1 -6706.508,E2 -6706.508} C_VEL
LIN {X 0,Y 482.655,Z 756.767,A -85,B 0,C 180,E1 -6706.953,E2 -6706.953} C_VEL
LIN {X 0,Y 483.085,Z 745.095,A -85,B 0,C 180,E1 -6707.898,E2 -6707.898} C_VEL
LIN {X 0,Y 483.537,Z 733.388,A -85,B 0,C 180,E1 -6708.633,E2 -6708.633} C_VEL
LIN {X 0,Y 483.882,Z 721.758,A -85,B 0,C 180,E1 -6709.189,E2 -6709.189} C_VEL
LIN {X 0,Y 484.128,Z 708.628,A -85,B 0,C 180,E1 -6709.638,E2 -6709.638} C_VEL
LIN {X 0,Y 484.309,Z 695.023,A -85,B 0,C 180,E1 -6709.916,E2 -6709.916} C_VEL
LIN {X 0,Y 484.851,Z 608.826,A -85,B 0,C 180,E1 -6711.237,E2 -6711.237} C_VEL
LIN {X 0,Y 482.285,Z 596.502,A -85,B 0,C 180,E1 -6711.538,E2 -6711.538} C_VEL
LIN {X 0,Y 482.472,Z 590.856,A -85,B 0,C 180,E1 -6712.808,E2 -6712.808} C_VEL
LIN {X 0,Y 481.697,Z 585.485,A -85,B 0,C 180,E1 -6714.104,E2 -6714.104} C_VEL
LIN {X 0,Y 481.669,Z 585.484,A -85,B 0,C 180,E1 -6717.327,E2 -6717.327} C_VEL
LIN {X 0,Y 481.675,Z 585.485,A -85,B 0,C 180,E1 -6720.26,E2 -6720.26} C_VEL
LIN {X 0,Y 481.743,Z 585.472,A -85,B 0,C 180,E1 -6723.113,E2 -6723.113} C_VEL
LIN {X 0,Y 481.676,Z 585.486,A -85,B 0,C 180,E1 -6725.888,E2 -6725.888} C_VEL
LIN {X 0,Y 481.701,Z 585.477,A -85,B 0,C 180,E1 -6729.028,E2 -6729.028} C_VEL
LIN {X 0,Y 481.707,Z 585.484,A -85,B 0,C 180,E1 -6732.16,E2 -6732.16} C_VEL
LIN {X 0,Y 481.742,Z 585.474,A -85,B 0,C 180,E1 -6734.777,E2 -6734.777} C_VEL
LIN {X 0,Y 481.795,Z 585.472,A -85,B 0,C 180,E1 -6738.217,E2 -6738.217} C_VEL
LIN {X 0,Y 481.763,Z 585.469,A -85,B 0,C 180,E1 -6741.613,E2 -6741.613} C_VEL
LIN {X 0,Y 481.817,Z 585.467,A -85,B 0,C 180,E1 -6744.141,E2 -6744.141} C_VEL
LIN {X 0,Y 481.93,Z 585.448,A -85,B 0,C 180,E1 -6747.493,E2 -6747.493} C_VEL
LIN {X 0,Y 481.907,Z 585.456,A -85,B 0,C 180,E1 -6750.837,E2 -6750.837} C_VEL
LIN {X 0,Y 481.931,Z 585.456,A -85,B 0,C 180,E1 -6752.508,E2 -6752.508} C_VEL
LIN {X 0,Y 481.819,Z 585.462,A -85,B 0,C 180,E1 -6755.861,E2 -6755.861} C_VEL
LIN {X 0,Y 481.766,Z 585.473,A -85,B 0,C 180,E1 -6758.389,E2 -6758.389} C_VEL
LIN {X 0,Y 481.754,Z 585.47,A -85,B 0,C 180,E1 -6761.786,E2 -6761.786} C_VEL
LIN {X 0,Y 481.746,Z 585.475,A -85,B 0,C 180,E1 -6765.225,E2 -6765.225} C_VEL
LIN {X 0,Y 481.715,Z 585.482,A -85,B 0,C 180,E1 -6768.722,E2 -6768.722} C_VEL
LIN {X 0,Y 481.649,Z 585.486,A -85,B 0,C 180,E1 -6771.395,E2 -6771.395} C_VEL
LIN {X 0,Y 481.677,Z 585.48,A -85,B 0,C 180,E1 -6774.114,E2 -6774.114} C_VEL
LIN {X 0,Y 481.751,Z 585.478,A -85,B 0,C 180,E1 -6777.14,E2 -6777.14} C_VEL
LIN {X 0,Y 481.683,Z 585.48,A -85,B 0,C 180,E1 -6779.742,E2 -6779.742} C_VEL
LIN {X 0,Y 481.676,Z 585.483,A -85,B 0,C 180,E1 -6782.675,E2 -6782.675} C_VEL
LIN {X 0,Y 481.641,Z 585.486,A -85,B 0,C 180,E1 -6785.71,E2 -6785.71} C_VEL
LIN {X 0,Y 481.675,Z 585.483,A -85,B 0,C 180,E1 -6788.86,E2 -6788.86} C_VEL
LIN {X 0,Y 481.656,Z 585.484,A -85,B 0,C 180,E1 -6791.913,E2 -6791.913} C_VEL
LIN {X 0,Y 481.659,Z 585.482,A -85,B 0,C 180,E1 -6794.458,E2 -6794.458} C_VEL
LIN {X 0,Y 481.652,Z 585.486,A -85,B 0,C 180,E1 -6797.84,E2 -6797.84} C_VEL
LIN {X 0,Y 481.665,Z 585.482,A -85,B 0,C 180,E1 -6800.654,E2 -6800.654} C_VEL
LIN {X 0,Y 481.632,Z 585.492,A -85,B 0,C 180,E1 -6803.377,E2 -6803.377} C_VEL
LIN {X 0,Y 481.714,Z 585.476,A -85,B 0,C 180,E1 -6806.33,E2 -6806.33} C_VEL
LIN {X 0,Y 481.655,Z 585.488,A -85,B 0,C 180,E1 -6809.418,E2 -6809.418} C_VEL
LIN {X 0,Y 481.705,Z 585.479,A -85,B 0,C 180,E1 -6812.168,E2 -6812.168} C_VEL
LIN {X 0,Y 481.698,Z 585.478,A -85,B 0,C 180,E1 -6814.969,E2 -6814.969} C_VEL
LIN {X 0,Y 481.654,Z 585.491,A -85,B 0,C 180,E1 -6817.705,E2 -6817.705} C_VEL
LIN {X 0,Y 481.709,Z 585.478,A -85,B 0,C 180,E1 -6820.393,E2 -6820.393} C_VEL
LIN {X 0,Y 481.684,Z 585.479,A -85,B 0,C 180,E1 -6823.034,E2 -6823.034} C_VEL
LIN {X 0,Y 481.695,Z 585.482,A -85,B 0,C 180,E1 -6825.639,E2 -6825.639} C_VEL
LIN {X 0,Y 481.756,Z 585.475,A -85,B 0,C 180,E1 -6828.215,E2 -6828.215} C_VEL
LIN {X 0,Y 481.766,Z 585.472,A -85,B 0,C 180,E1 -6831.612,E2 -6831.612} C_VEL
LIN {X 0,Y 481.816,Z 585.471,A -85,B 0,C 180,E1 -6834.14,E2 -6834.14} C_VEL
LIN {X 0,Y 481.933,Z 585.449,A -85,B 0,C 180,E1 -6837.493,E2 -6837.493} C_VEL
LIN {X 0,Y 481.891,Z 585.454,A -85,B 0,C 180,E1 -6840.836,E2 -6840.836} C_VEL
LIN {X 0,Y 481.933,Z 585.453,A -85,B 0,C 180,E1 -6842.508,E2 -6842.508} C_VEL
LIN {X 0,Y 481.82,Z 585.465,A -85,B 0,C 180,E1 -6845.86,E2 -6845.86} C_VEL
LIN {X 0,Y 481.767,Z 585.477,A -85,B 0,C 180,E1 -6848.388,E2 -6848.388} C_VEL
LIN {X 0,Y 481.757,Z 585.471,A -85,B 0,C 180,E1 -6851.785,E2 -6851.785} C_VEL
LIN {X 0,Y 481.748,Z 585.471,A -85,B 0,C 180,E1 -6855.224,E2 -6855.224} C_VEL
LIN {X 0,Y 481.714,Z 585.481,A -85,B 0,C 180,E1 -6858.722,E2 -6858.722} C_VEL
LIN {X 0,Y 481.651,Z 585.483,A -85,B 0,C 180,E1 -6861.395,E2 -6861.395} C_VEL
LIN {X 0,Y 481.679,Z 585.482,A -85,B 0,C 180,E1 -6864.113,E2 -6864.113} C_VEL
LIN {X 0,Y 481.752,Z 585.473,A -85,B 0,C 180,E1 -6867.139,E2 -6867.139} C_VEL
LIN {X 0,Y 481.684,Z 585.479,A -85,B 0,C 180,E1 -6869.741,E2 -6869.741} C_VEL
LIN {X 0,Y 481.678,Z 585.487,A -85,B 0,C 180,E1 -6872.674,E2 -6872.674} C_VEL
LIN {X 0,Y 481.643,Z 585.484,A -85,B 0,C 180,E1 -6875.709,E2 -6875.709} C_VEL
LIN {X 0,Y 481.676,Z 585.489,A -85,B 0,C 180,E1 -6878.859,E2 -6878.859} C_VEL
LIN {X 0,Y 481.658,Z 585.482,A -85,B 0,C 180,E1 -6881.913,E2 -6881.913} C_VEL
LIN {X 0,Y 481.665,Z 585.483,A -85,B 0,C 180,E1 -6884.457,E2 -6884.457} C_VEL
LIN {X 0,Y 481.653,Z 585.483,A -85,B 0,C 180,E1 -6887.839,E2 -6887.839} C_VEL
LIN {X 0,Y 481.686,Z 585.481,A -85,B 0,C 180,E1 -6890.651,E2 -6890.651} C_VEL
LIN {X 0,Y 481.633,Z 585.491,A -85,B 0,C 180,E1 -6893.376,E2 -6893.376} C_VEL
LIN {X 0,Y 481.715,Z 585.477,A -85,B 0,C 180,E1 -6896.33,E2 -6896.33} C_VEL
LIN {X 0,Y 481.655,Z 585.49,A -85,B 0,C 180,E1 -6899.417,E2 -6899.417} C_VEL
LIN {X 0,Y 481.705,Z 585.481,A -85,B 0,C 180,E1 -6902.168,E2 -6902.168} C_VEL
LIN {X 0,Y 481.767,Z 585.632,A -85,B 0,C 180,E1 -6903.171,E2 -6903.171} C_VEL
LIN {X 0,Y 484.19,Z 597.852,A -85,B 0,C 180,E1 -6905.335,E2 -6905.335} C_VEL
LIN {X 0,Y 483.87,Z 610.275,A -85,B 0,C 180,E1 -6907.362,E2 -6907.362} C_VEL
LIN {X 0,Y 483.043,Z 630.789,A -85,B 0,C 180,E1 -6910.643,E2 -6910.643} C_VEL
LIN {X 0,Y 482.399,Z 648.861,A -85,B 0,C 180,E1 -6913.492,E2 -6913.492} C_VEL
LIN {X 0,Y 484.798,Z 666.251,A -85,B 0,C 180,E1 -6913.847,E2 -6913.847} C_VEL
LIN {X 0,Y 484.159,Z 757.623,A -85,B 0,C 180,E1 -6915.256,E2 -6915.256} C_VEL
LIN {X 0,Y 483.796,Z 770.828,A -85,B 0,C 180,E1 -6915.621,E2 -6915.621} C_VEL
LIN {X 0,Y 483.435,Z 784.119,A -85,B 0,C 180,E1 -6916.174,E2 -6916.174} C_VEL
LIN {X 0,Y 482.979,Z 796.572,A -85,B 0,C 180,E1 -6916.889,E2 -6916.889} C_VEL
LIN {X 0,Y 482.567,Z 807.593,A -85,B 0,C 180,E1 -6917.701,E2 -6917.701} C_VEL
LIN {X 0,Y 482.159,Z 817.971,A -85,B 0,C 180,E1 -6918.651,E2 -6918.651} C_VEL
LIN {X 0,Y 481.752,Z 827.287,A -85,B 0,C 180,E1 -6919.705,E2 -6919.705} C_VEL
LIN {X 0,Y 481.39,Z 836.343,A -85,B 0,C 180,E1 -6920.97,E2 -6920.97} C_VEL
LIN {X 0,Y 481.15,Z 843.639,A -85,B 0,C 180,E1 -6922.234,E2 -6922.234} C_VEL
LIN {X 0,Y 480.952,Z 849.666,A -85,B 0,C 180,E1 -6923.548,E2 -6923.548} C_VEL
LIN {X 0,Y 480.905,Z 854.683,A -85,B 0,C 180,E1 -6924.969,E2 -6924.969} C_VEL
LIN {X 0,Y 480.851,Z 857.004,A -85,B 0,C 180,E1 -6925.808,E2 -6925.808} C_VEL
LIN {X 0,Y 480.892,Z 858.893,A -85,B 0,C 180,E1 -6926.648,E2 -6926.648} C_VEL
LIN {X 0,Y 480.869,Z 860.306,A -85,B 0,C 180,E1 -6927.486,E2 -6927.486} C_VEL
LIN {X 0,Y 480.824,Z 861.308,A -85,B 0,C 180,E1 -6928.324,E2 -6928.324} C_VEL
LIN {X 0,Y 480.743,Z 862.126,A -85,B 0,C 180,E1 -6929.999,E2 -6929.999} C_VEL
LIN {X 0,Y 480.825,Z 861.281,A -85,B 0,C 180,E1 -6931.674,E2 -6931.674} C_VEL
LIN {X 0,Y 480.88,Z 860.263,A -85,B 0,C 180,E1 -6932.512,E2 -6932.512} C_VEL
LIN {X 0,Y 480.892,Z 858.834,A -85,B 0,C 180,E1 -6933.35,E2 -6933.35} C_VEL
LIN {X 0,Y 480.852,Z 855.835,A -85,B 0,C 180,E1 -6934.61,E2 -6934.61} C_VEL
LIN {X 0,Y 480.95,Z 851.786,A -85,B 0,C 180,E1 -6935.87,E2 -6935.87} C_VEL
LIN {X 0,Y 481.108,Z 845.558,A -85,B 0,C 180,E1 -6937.343,E2 -6937.343} C_VEL
LIN {X 0,Y 481.32,Z 838.755,A -85,B 0,C 180,E1 -6938.607,E2 -6938.607} C_VEL
LIN {X 0,Y 481.59,Z 830.316,A -85,B 0,C 180,E1 -6939.872,E2 -6939.872} C_VEL
LIN {X 0,Y 481.923,Z 821.642,A -85,B 0,C 180,E1 -6940.927,E2 -6940.927} C_VEL
LIN {X 0,Y 482.284,Z 812.143,A -85,B 0,C 180,E1 -6941.876,E2 -6941.876} C_VEL
LIN {X 0,Y 482.795,Z 800.642,A -85,B 0,C 180,E1 -6942.804,E2 -6942.804} C_VEL
LIN {X 0,Y 483.182,Z 788.656,A -85,B 0,C 180,E1 -6943.564,E2 -6943.564} C_VEL
LIN {X 0,Y 483.618,Z 776.53,A -85,B 0,C 180,E1 -6944.141,E2 -6944.141} C_VEL
LIN {X 0,Y 483.996,Z 764.324,A -85,B 0,C 180,E1 -6944.559,E2 -6944.559} C_VEL
LIN {X 0,Y 484.185,Z 750.973,A -85,B 0,C 180,E1 -6944.849,E2 -6944.849} C_VEL
LIN {X 0,Y 484.721,Z 664.773,A -85,B 0,C 180,E1 -6946.168,E2 -6946.168} C_VEL
LIN {X 0,Y 482.364,Z 648.004,A -85,B 0,C 180,E1 -6946.532,E2 -6946.532} C_VEL
LIN {X 0,Y 483.017,Z 627.396,A -85,B 0,C 180,E1 -6949.772,E2 -6949.772} C_VEL
LIN {X 0,Y 483.735,Z 609.392,A -85,B 0,C 180,E1 -6952.643,E2 -6952.643} C_VEL
LIN {X 0,Y 484.149,Z 598.333,A -85,B 0,C 180,E1 -6954.437,E2 -6954.437} C_VEL
LIN {X 0,Y 482.388,Z 588.571,A -85,B 0,C 180,E1 -6956.148,E2 -6956.148} C_VEL
LIN {X 0,Y 481.745,Z 585.48,A -85,B 0,C 180,E1 -6956.711,E2 -6956.711} C_VEL
LIN {X 0,Y 481.677,Z 585.484,A -85,B 0,C 180,E1 -6959.74,E2 -6959.74} C_VEL
LIN {X 0,Y 481.67,Z 585.49,A -85,B 0,C 180,E1 -6962.673,E2 -6962.673} C_VEL
LIN {X 0,Y 481.64,Z 585.488,A -85,B 0,C 180,E1 -6965.708,E2 -6965.708} C_VEL
LIN {X 0,Y 481.711,Z 585.479,A -85,B 0,C 180,E1 -6969.353,E2 -6969.353} C_VEL
LIN {X 0,Y 481.644,Z 585.492,A -85,B 0,C 180,E1 -6972.159,E2 -6972.159} C_VEL
LIN {X 0,Y 481.655,Z 585.486,A -85,B 0,C 180,E1 -6975.542,E2 -6975.542} C_VEL
LIN {X 0,Y 481.668,Z 585.487,A -85,B 0,C 180,E1 -6978.083,E2 -6978.083} C_VEL
LIN {X 0,Y 481.699,Z 585.479,A -85,B 0,C 180,E1 -6981.143,E2 -6981.143} C_VEL
LIN {X 0,Y 481.663,Z 585.486,A -85,B 0,C 180,E1 -6984.794,E2 -6984.794} C_VEL
LIN {X 0,Y 481.667,Z 585.482,A -85,B 0,C 180,E1 -6987.325,E2 -6987.325} C_VEL
LIN {X 0,Y 481.682,Z 585.485,A -85,B 0,C 180,E1 -6990.259,E2 -6990.259} C_VEL
LIN {X 0,Y 481.745,Z 585.472,A -85,B 0,C 180,E1 -6993.112,E2 -6993.112} C_VEL
LIN {X 0,Y 481.67,Z 585.483,A -85,B 0,C 180,E1 -6995.886,E2 -6995.886} C_VEL
LIN {X 0,Y 481.694,Z 585.478,A -85,B 0,C 180,E1 -6999.027,E2 -6999.027} C_VEL
LIN {X 0,Y 481.7,Z 585.484,A -85,B 0,C 180,E1 -7002.158,E2 -7002.158} C_VEL
LIN {X 0,Y 481.734,Z 585.476,A -85,B 0,C 180,E1 -7004.775,E2 -7004.775} C_VEL
LIN {X 0,Y 481.787,Z 585.472,A -85,B 0,C 180,E1 -7008.216,E2 -7008.216} C_VEL
LIN {X 0,Y 481.755,Z 585.473,A -85,B 0,C 180,E1 -7011.611,E2 -7011.611} C_VEL
LIN {X 0,Y 481.809,Z 585.471,A -85,B 0,C 180,E1 -7014.139,E2 -7014.139} C_VEL
LIN {X 0,Y 481.921,Z 585.451,A -85,B 0,C 180,E1 -7017.492,E2 -7017.492} C_VEL
LIN {X 0,Y 481.932,Z 585.454,A -85,B 0,C 180,E1 -7020,E2 -7020} C_VEL
LIN {X 0,Y 481.921,Z 585.458,A -85,B 0,C 180,E1 -7022.507,E2 -7022.507} C_VEL
LIN {X 0,Y 481.823,Z 585.468,A -85,B 0,C 180,E1 -7025.86,E2 -7025.86} C_VEL
LIN {X 0,Y 481.756,Z 585.479,A -85,B 0,C 180,E1 -7028.388,E2 -7028.388} C_VEL
LIN {X 0,Y 481.787,Z 585.471,A -85,B 0,C 180,E1 -7031.784,E2 -7031.784} C_VEL
LIN {X 0,Y 481.749,Z 585.481,A -85,B 0,C 180,E1 -7035.754,E2 -7035.754} C_VEL
LIN {X 0,Y 482.512,Z 590.328,A -85,B 0,C 180,E1 -7036.936,E2 -7036.936} C_VEL
LIN {X 0,Y 482.439,Z 597.53,A -85,B 0,C 180,E1 -7038.576,E2 -7038.576} C_VEL
LIN {X 0,Y 485.01,Z 609.762,A -85,B 0,C 180,E1 -7038.864,E2 -7038.864} C_VEL
LIN {X 0,Y 484.224,Z 703.685,A -85,B 0,C 180,E1 -7040.33,E2 -7040.33} C_VEL
LIN {X 0,Y 483.961,Z 717.573,A -85,B 0,C 180,E1 -7040.73,E2 -7040.73} C_VEL
LIN {X 0,Y 483.644,Z 729.656,A -85,B 0,C 180,E1 -7041.246,E2 -7041.246} C_VEL
LIN {X 0,Y 483.326,Z 741.254,A -85,B 0,C 180,E1 -7041.916,E2 -7041.916} C_VEL
LIN {X 0,Y 482.896,Z 751.765,A -85,B 0,C 180,E1 -7042.686,E2 -7042.686} C_VEL
LIN {X 0,Y 482.426,Z 762.933,A -85,B 0,C 180,E1 -7043.708,E2 -7043.708} C_VEL
LIN {X 0,Y 482.04,Z 772.273,A -85,B 0,C 180,E1 -7044.782,E2 -7044.782} C_VEL
LIN {X 0,Y 481.628,Z 780.622,A -85,B 0,C 180,E1 -7045.961,E2 -7045.961} C_VEL
LIN {X 0,Y 481.414,Z 787.002,A -85,B 0,C 180,E1 -7047.064,E2 -7047.064} C_VEL
LIN {X 0,Y 481.222,Z 792.929,A -85,B 0,C 180,E1 -7048.324,E2 -7048.324} C_VEL
LIN {X 0,Y 480.999,Z 798.289,A -85,B 0,C 180,E1 -7049.787,E2 -7049.787} C_VEL
LIN {X 0,Y 480.913,Z 802.138,A -85,B 0,C 180,E1 -7051.251,E2 -7051.251} C_VEL
LIN {X 0,Y 480.779,Z 804.72,A -85,B 0,C 180,E1 -7052.742,E2 -7052.742} C_VEL
LIN {X 0,Y 480.76,Z 805.75,A -85,B 0,C 180,E1 -7053.745,E2 -7053.745} C_VEL
LIN {X 0,Y 480.76,Z 806.211,A -85,B 0,C 180,E1 -7055.053,E2 -7055.053} C_VEL
LIN {X 0,Y 480.747,Z 805.603,A -85,B 0,C 180,E1 -7056.484,E2 -7056.484} C_VEL
LIN {X 0,Y 480.781,Z 803.897,A -85,B 0,C 180,E1 -7057.876,E2 -7057.876} C_VEL
LIN {X 0,Y 480.904,Z 801.122,A -85,B 0,C 180,E1 -7059.238,E2 -7059.238} C_VEL
LIN {X 0,Y 481.069,Z 797.286,A -85,B 0,C 180,E1 -7060.566,E2 -7060.566} C_VEL
LIN {X 0,Y 481.153,Z 792.433,A -85,B 0,C 180,E1 -7061.848,E2 -7061.848} C_VEL
LIN {X 0,Y 481.416,Z 786.32,A -85,B 0,C 180,E1 -7063.121,E2 -7063.121} C_VEL
LIN {X 0,Y 481.711,Z 778.332,A -85,B 0,C 180,E1 -7064.451,E2 -7064.451} C_VEL
LIN {X 0,Y 482.093,Z 769.733,A -85,B 0,C 180,E1 -7065.595,E2 -7065.595} C_VEL
LIN {X 0,Y 482.466,Z 760.549,A -85,B 0,C 180,E1 -7066.595,E2 -7066.595} C_VEL
LIN {X 0,Y 482.655,Z 756.767,A -85,B 0,C 180,E1 -7066.953,E2 -7066.953} C_VEL
LIN {X 0,Y 482.196,Z 752.135,A -85,B 0,C 180,E1 -7067.375,E2 -7067.375} C_VEL
LIN {X 0,Y 479.684,Z 744.43,A -85,B 0,C 180,E1 -7068.049,E2 -7068.049} C_VEL
LIN {X 0,Y 477.243,Z 736.24,A -85,B 0,C 180,E1 -7068.661,E2 -7068.661} C_VEL
LIN {X 0,Y 476.74,Z 730.943,A -85,B 0,C 180,E1 -7068.976,E2 -7068.976} C_VEL
LIN {X 0,Y 477.079,Z 718.199,A -85,B 0,C 180,E1 -7069.545,E2 -7069.545} C_VEL
LIN {X 0,Y 477.309,Z 704.835,A -85,B 0,C 180,E1 -7069.947,E2 -7069.947} C_VEL
LIN {X 0,Y 477.598,Z 676.593,A -85,B 0,C 180,E1 -7070.415,E2 -7070.415} C_VEL
LIN {X 0,Y 478.027,Z 609.555,A -85,B 0,C 180,E1 -7071.465,E2 -7071.465} C_VEL
LIN {X 0,Y 475.335,Z 596.879,A -85,B 0,C 180,E1 -7071.783,E2 -7071.783} C_VEL
LIN {X 0,Y 475.465,Z 591.697,A -85,B 0,C 180,E1 -7072.958,E2 -7072.958} C_VEL
LIN {X 0,Y 474.659,Z 586.361,A -85,B 0,C 180,E1 -7074.259,E2 -7074.259} C_VEL
LIN {X 0,Y 474.612,Z 586.365,A -85,B 0,C 180,E1 -7077.57,E2 -7077.57} C_VEL
LIN {X 0,Y 474.62,Z 586.359,A -85,B 0,C 180,E1 -7080.886,E2 -7080.886} C_VEL
LIN {X 0,Y 474.658,Z 586.357,A -85,B 0,C 180,E1 -7083.629,E2 -7083.629} C_VEL
LIN {X 0,Y 474.634,Z 586.359,A -85,B 0,C 180,E1 -7086.642,E2 -7086.642} C_VEL
LIN {X 0,Y 474.656,Z 586.362,A -85,B 0,C 180,E1 -7090.091,E2 -7090.091} C_VEL
LIN {X 0,Y 474.651,Z 586.357,A -85,B 0,C 180,E1 -7092.776,E2 -7092.776} C_VEL
LIN {X 0,Y 474.648,Z 586.356,A -85,B 0,C 180,E1 -7095.422,E2 -7095.422} C_VEL
LIN {X 0,Y 474.739,Z 586.349,A -85,B 0,C 180,E1 -7098.039,E2 -7098.039} C_VEL
LIN {X 0,Y 474.728,Z 586.345,A -85,B 0,C 180,E1 -7101.487,E2 -7101.487} C_VEL
LIN {X 0,Y 474.779,Z 586.343,A -85,B 0,C 180,E1 -7104.053,E2 -7104.053} C_VEL
LIN {X 0,Y 474.896,Z 586.325,A -85,B 0,C 180,E1 -7107.456,E2 -7107.456} C_VEL
LIN {X 0,Y 474.913,Z 586.324,A -85,B 0,C 180,E1 -7110.001,E2 -7110.001} C_VEL
LIN {X 0,Y 474.897,Z 586.333,A -85,B 0,C 180,E1 -7112.546,E2 -7112.546} C_VEL
LIN {X 0,Y 474.781,Z 586.34,A -85,B 0,C 180,E1 -7115.948,E2 -7115.948} C_VEL
LIN {X 0,Y 474.731,Z 586.351,A -85,B 0,C 180,E1 -7118.514,E2 -7118.514} C_VEL
LIN {X 0,Y 474.707,Z 586.348,A -85,B 0,C 180,E1 -7121.963,E2 -7121.963} C_VEL
LIN {X 0,Y 474.703,Z 586.35,A -85,B 0,C 180,E1 -7125.456,E2 -7125.456} C_VEL
LIN {X 0,Y 474.668,Z 586.36,A -85,B 0,C 180,E1 -7129.011,E2 -7129.011} C_VEL
LIN {X 0,Y 474.592,Z 586.363,A -85,B 0,C 180,E1 -7131.73,E2 -7131.73} C_VEL
LIN {X 0,Y 474.66,Z 586.356,A -85,B 0,C 180,E1 -7134.494,E2 -7134.494} C_VEL
LIN {X 0,Y 474.685,Z 586.356,A -85,B 0,C 180,E1 -7137.335,E2 -7137.335} C_VEL
LIN {X 0,Y 474.609,Z 586.36,A -85,B 0,C 180,E1 -7140.231,E2 -7140.231} C_VEL
LIN {X 0,Y 474.647,Z 586.364,A -85,B 0,C 180,E1 -7143.221,E2 -7143.221} C_VEL
LIN {X 0,Y 474.593,Z 586.362,A -85,B 0,C 180,E1 -7146.324,E2 -7146.324} C_VEL
LIN {X 0,Y 474.632,Z 586.361,A -85,B 0,C 180,E1 -7149.648,E2 -7149.648} C_VEL
LIN {X 0,Y 474.618,Z 586.362,A -85,B 0,C 180,E1 -7152.935,E2 -7152.935} C_VEL
LIN {X 0,Y 474.61,Z 586.362,A -85,B 0,C 180,E1 -7155.895,E2 -7155.895} C_VEL
LIN {X 0,Y 474.632,Z 586.361,A -85,B 0,C 180,E1 -7159.041,E2 -7159.041} C_VEL
LIN {X 0,Y 474.614,Z 586.365,A -85,B 0,C 180,E1 -7161.705,E2 -7161.705} C_VEL
LIN {X 0,Y 474.629,Z 586.358,A -85,B 0,C 180,E1 -7164.726,E2 -7164.726} C_VEL
LIN {X 0,Y 474.64,Z 586.363,A -85,B 0,C 180,E1 -7167.788,E2 -7167.788} C_VEL
LIN {X 0,Y 474.628,Z 586.358,A -85,B 0,C 180,E1 -7170.885,E2 -7170.885} C_VEL
LIN {X 0,Y 474.659,Z 586.362,A -85,B 0,C 180,E1 -7173.628,E2 -7173.628} C_VEL
LIN {X 0,Y 474.639,Z 586.357,A -85,B 0,C 180,E1 -7176.642,E2 -7176.642} C_VEL
LIN {X 0,Y 474.659,Z 586.359,A -85,B 0,C 180,E1 -7180.09,E2 -7180.09} C_VEL
LIN {X 0,Y 474.644,Z 586.356,A -85,B 0,C 180,E1 -7182.774,E2 -7182.774} C_VEL
LIN {X 0,Y 474.653,Z 586.357,A -85,B 0,C 180,E1 -7185.421,E2 -7185.421} C_VEL
LIN {X 0,Y 474.71,Z 586.356,A -85,B 0,C 180,E1 -7188.038,E2 -7188.038} C_VEL
LIN {X 0,Y 474.732,Z 586.347,A -85,B 0,C 180,E1 -7191.487,E2 -7191.487} C_VEL
LIN {X 0,Y 474.778,Z 586.348,A -85,B 0,C 180,E1 -7194.053,E2 -7194.053} C_VEL
LIN {X 0,Y 474.899,Z 586.325,A -85,B 0,C 180,E1 -7197.456,E2 -7197.456} C_VEL
LIN {X 0,Y 474.917,Z 586.328,A -85,B 0,C 180,E1 -7200,E2 -7200} C_VEL
LIN {X 0,Y 474.899,Z 586.329,A -85,B 0,C 180,E1 -7202.545,E2 -7202.545} C_VEL
LIN {X 0,Y 474.783,Z 586.342,A -85,B 0,C 180,E1 -7205.948,E2 -7205.948} C_VEL
LIN {X 0,Y 474.732,Z 586.351,A -85,B 0,C 180,E1 -7208.514,E2 -7208.514} C_VEL
LIN {X 0,Y 474.71,Z 586.351,A -85,B 0,C 180,E1 -7211.962,E2 -7211.962} C_VEL
LIN {X 0,Y 474.705,Z 586.348,A -85,B 0,C 180,E1 -7215.456,E2 -7215.456} C_VEL
LIN {X 0,Y 474.668,Z 586.355,A -85,B 0,C 180,E1 -7219.01,E2 -7219.01} C_VEL
LIN {X 0,Y 474.594,Z 586.362,A -85,B 0,C 180,E1 -7221.729,E2 -7221.729} C_VEL
LIN {X 0,Y 474.661,Z 586.361,A -85,B 0,C 180,E1 -7224.493,E2 -7224.493} C_VEL
LIN {X 0,Y 474.687,Z 586.352,A -85,B 0,C 180,E1 -7227.334,E2 -7227.334} C_VEL
LIN {X 0,Y 474.611,Z 586.362,A -85,B 0,C 180,E1 -7230.23,E2 -7230.23} C_VEL
LIN {X 0,Y 474.648,Z 586.358,A -85,B 0,C 180,E1 -7233.22,E2 -7233.22} C_VEL
LIN {X 0,Y 474.594,Z 586.364,A -85,B 0,C 180,E1 -7236.323,E2 -7236.323} C_VEL
LIN {X 0,Y 474.623,Z 586.359,A -85,B 0,C 180,E1 -7239.646,E2 -7239.646} C_VEL
LIN {X 0,Y 474.621,Z 586.367,A -85,B 0,C 180,E1 -7242.934,E2 -7242.934} C_VEL
LIN {X 0,Y 474.615,Z 586.36,A -85,B 0,C 180,E1 -7245.895,E2 -7245.895} C_VEL
LIN {X 0,Y 474.633,Z 586.366,A -85,B 0,C 180,E1 -7249.04,E2 -7249.04} C_VEL
LIN {X 0,Y 474.615,Z 586.361,A -85,B 0,C 180,E1 -7251.704,E2 -7251.704} C_VEL
LIN {X 0,Y 474.631,Z 586.36,A -85,B 0,C 180,E1 -7254.725,E2 -7254.725} C_VEL
LIN {X 0,Y 474.641,Z 586.36,A -85,B 0,C 180,E1 -7257.787,E2 -7257.787} C_VEL
LIN {X 0,Y 474.629,Z 586.364,A -85,B 0,C 180,E1 -7260.884,E2 -7260.884} C_VEL
LIN {X 0,Y 474.741,Z 586.481,A -85,B 0,C 180,E1 -7262.95,E2 -7262.95} C_VEL
LIN {X 0,Y 477.22,Z 598.896,A -85,B 0,C 180,E1 -7265.182,E2 -7265.182} C_VEL
LIN {X 0,Y 477.08,Z 607.18,A -85,B 0,C 180,E1 -7266.562,E2 -7266.562} C_VEL
LIN {X 0,Y 476.26,Z 625.069,A -85,B 0,C 180,E1 -7269.483,E2 -7269.483} C_VEL
LIN {X 0,Y 475.6,Z 642.97,A -85,B 0,C 180,E1 -7272.365,E2 -7272.365} C_VEL
LIN {X 0,Y 475.455,Z 648.675,A -85,B 0,C 180,E1 -7273.248,E2 -7273.248} C_VEL
LIN {X 0,Y 477.982,Z 666.831,A -85,B 0,C 180,E1 -7273.626,E2 -7273.626} C_VEL
LIN {X 0,Y 477.273,Z 758.042,A -85,B 0,C 180,E1 -7275.066,E2 -7275.066} C_VEL
LIN {X 0,Y 476.85,Z 771.729,A -85,B 0,C 180,E1 -7275.462,E2 -7275.462} C_VEL
LIN {X 0,Y 476.468,Z 784.602,A -85,B 0,C 180,E1 -7276.022,E2 -7276.022} C_VEL
LIN {X 0,Y 476.012,Z 796.056,A -85,B 0,C 180,E1 -7276.694,E2 -7276.694} C_VEL
LIN {X 0,Y 475.594,Z 807.006,A -85,B 0,C 180,E1 -7277.51,E2 -7277.51} C_VEL
LIN {X 0,Y 475.174,Z 817.499,A -85,B 0,C 180,E1 -7278.481,E2 -7278.481} C_VEL
LIN {X 0,Y 474.717,Z 826.832,A -85,B 0,C 180,E1 -7279.55,E2 -7279.55} C_VEL
LIN {X 0,Y 474.34,Z 835.9,A -85,B 0,C 180,E1 -7280.834,E2 -7280.834} C_VEL
LIN {X 0,Y 474.074,Z 843.205,A -85,B 0,C 180,E1 -7282.117,E2 -7282.117} C_VEL
LIN {X 0,Y 473.927,Z 848.138,A -85,B 0,C 180,E1 -7283.186,E2 -7283.186} C_VEL
LIN {X 0,Y 473.874,Z 852.933,A -85,B 0,C 180,E1 -7284.467,E2 -7284.467} C_VEL
LIN {X 0,Y 473.755,Z 856.589,A -85,B 0,C 180,E1 -7285.745,E2 -7285.745} C_VEL
LIN {X 0,Y 473.818,Z 858.482,A -85,B 0,C 180,E1 -7286.598,E2 -7286.598} C_VEL
LIN {X 0,Y 473.783,Z 859.896,A -85,B 0,C 180,E1 -7287.449,E2 -7287.449} C_VEL
LIN {X 0,Y 473.758,Z 860.899,A -85,B 0,C 180,E1 -7288.299,E2 -7288.299} C_VEL
LIN {X 0,Y 473.669,Z 861.715,A -85,B 0,C 180,E1 -7289.999,E2 -7289.999} C_VEL
LIN {X 0,Y 473.688,Z 861.489,A -85,B 0,C 180,E1 -7290.849,E2 -7290.849} C_VEL
LIN {X 0,Y 473.758,Z 860.864,A -85,B 0,C 180,E1 -7291.699,E2 -7291.699} C_VEL
LIN {X 0,Y 473.793,Z 859.841,A -85,B 0,C 180,E1 -7292.55,E2 -7292.55} C_VEL
LIN {X 0,Y 473.818,Z 858.409,A -85,B 0,C 180,E1 -7293.4,E2 -7293.4} C_VEL
LIN {X 0,Y 473.774,Z 855.4,A -85,B 0,C 180,E1 -7294.679,E2 -7294.679} C_VEL
LIN {X 0,Y 473.853,Z 851.339,A -85,B 0,C 180,E1 -7295.958,E2 -7295.958} C_VEL
LIN {X 0,Y 474.017,Z 845.092,A -85,B 0,C 180,E1 -7297.453,E2 -7297.453} C_VEL
LIN {X 0,Y 474.246,Z 838.274,A -85,B 0,C 180,E1 -7298.736,E2 -7298.736} C_VEL
LIN {X 0,Y 474.533,Z 829.817,A -85,B 0,C 180,E1 -7300.021,E2 -7300.021} C_VEL
LIN {X 0,Y 474.913,Z 821.12,A -85,B 0,C 180,E1 -7301.091,E2 -7301.091} C_VEL
LIN {X 0,Y 475.358,Z 810.662,A -85,B 0,C 180,E1 -7302.138,E2 -7302.138} C_VEL
LIN {X 0,Y 475.863,Z 799.792,A -85,B 0,C 180,E1 -7303.015,E2 -7303.015} C_VEL
LIN {X 0,Y 476.266,Z 788.058,A -85,B 0,C 180,E1 -7303.764,E2 -7303.764} C_VEL
LIN {X 0,Y 476.722,Z 775.896,A -85,B 0,C 180,E1 -7304.35,E2 -7304.35} C_VEL
LIN {X 0,Y 477.079,Z 764.543,A -85,B 0,C 180,E1 -7304.747,E2 -7304.747} C_VEL
LIN {X 0,Y 477.303,Z 751.704,A -85,B 0,C 180,E1 -7305.04,E2 -7305.04} C_VEL
LIN {X 0,Y 477.929,Z 665.882,A -85,B 0,C 180,E1 -7306.379,E2 -7306.379} C_VEL
LIN {X 0,Y 475.363,Z 647.55,A -85,B 0,C 180,E1 -7306.783,E2 -7306.783} C_VEL
LIN {X 0,Y 476.088,Z 626.985,A -85,B 0,C 180,E1 -7310.072,E2 -7310.072} C_VEL
LIN {X 0,Y 476.795,Z 609.03,A -85,B 0,C 180,E1 -7312.991,E2 -7312.991} C_VEL
LIN {X 0,Y 477.208,Z 599.369,A -85,B 0,C 180,E1 -7314.584,E2 -7314.584} C_VEL
LIN {X 0,Y 474.715,Z 586.361,A -85,B 0,C 180,E1 -7316.931,E2 -7316.931} C_VEL
LIN {X 0,Y 474.603,Z 586.37,A -85,B 0,C 180,E1 -7320.229,E2 -7320.229} C_VEL
LIN {X 0,Y 474.64,Z 586.361,A -85,B 0,C 180,E1 -7323.219,E2 -7323.219} C_VEL
LIN {X 0,Y 474.591,Z 586.37,A -85,B 0,C 180,E1 -7326.322,E2 -7326.322} C_VEL
LIN {X 0,Y 474.647,Z 586.359,A -85,B 0,C 180,E1 -7329.65,E2 -7329.65} C_VEL
LIN {X 0,Y 474.61,Z 586.367,A -85,B 0,C 180,E1 -7332.933,E2 -7332.933} C_VEL
LIN {X 0,Y 474.613,Z 586.365,A -85,B 0,C 180,E1 -7335.895,E2 -7335.895} C_VEL
LIN {X 0,Y 474.64,Z 586.36,A -85,B 0,C 180,E1 -7339.037,E2 -7339.037} C_VEL
LIN {X 0,Y 474.615,Z 586.361,A -85,B 0,C 180,E1 -7341.701,E2 -7341.701} C_VEL
LIN {X 0,Y 474.624,Z 586.364,A -85,B 0,C 180,E1 -7344.725,E2 -7344.725} C_VEL
LIN {X 0,Y 474.631,Z 586.359,A -85,B 0,C 180,E1 -7347.787,E2 -7347.787} C_VEL
LIN {X 0,Y 474.625,Z 586.359,A -85,B 0,C 180,E1 -7350.882,E2 -7350.882} C_VEL
LIN {X 0,Y 474.659,Z 586.354,A -85,B 0,C 180,E1 -7353.628,E2 -7353.628} C_VEL
LIN {X 0,Y 474.628,Z 586.362,A -85,B 0,C 180,E1 -7356.641,E2 -7356.641} C_VEL
LIN {X 0,Y 474.649,Z 586.359,A -85,B 0,C 180,E1 -7360.089,E2 -7360.089} C_VEL
LIN {X 0,Y 474.643,Z 586.361,A -85,B 0,C 180,E1 -7362.774,E2 -7362.774} C_VEL
LIN {X 0,Y 474.64,Z 586.356,A -85,B 0,C 180,E1 -7365.421,E2 -7365.421} C_VEL
LIN {X 0,Y 474.731,Z 586.35,A -85,B 0,C 180,E1 -7368.038,E2 -7368.038} C_VEL
LIN {X 0,Y 474.72,Z 586.349,A -85,B 0,C 180,E1 -7371.486,E2 -7371.486} C_VEL
LIN {X 0,Y 474.771,Z 586.346,A -85,B 0,C 180,E1 -7374.052,E2 -7374.052} C_VEL
LIN {X 0,Y 474.887,Z 586.328,A -85,B 0,C 180,E1 -7377.455,E2 -7377.455} C_VEL
LIN {X 0,Y 474.868,Z 586.332,A -85,B 0,C 180,E1 -7380.848,E2 -7380.848} C_VEL
LIN {X 0,Y 474.887,Z 586.334,A -85,B 0,C 180,E1 -7382.545,E2 -7382.545} C_VEL
LIN {X 0,Y 474.783,Z 586.346,A -85,B 0,C 180,E1 -7385.947,E2 -7385.947} C_VEL
LIN {X 0,Y 474.721,Z 586.355,A -85,B 0,C 180,E1 -7388.514,E2 -7388.514} C_VEL
LIN {X 0,Y 474.731,Z 586.353,A -85,B 0,C 180,E1 -7391.962,E2 -7391.962} C_VEL
LIN {X 0,Y 474.747,Z 586.533,A -85,B 0,C 180,E1 -7395.604,E2 -7395.604} C_VEL
LIN {X 0,Y 475.59,Z 593.021,A -85,B 0,C 180,E1 -7397.19,E2 -7397.19} C_VEL
LIN {X 0,Y 475.483,Z 597.82,A -85,B 0,C 180,E1 -7398.311,E2 -7398.311} C_VEL
LIN {X 0,Y 478.185,Z 610.506,A -85,B 0,C 180,E1 -7398.631,E2 -7398.631} C_VEL
LIN {X 0,Y 477.374,Z 704.466,A -85,B 0,C 180,E1 -7400.129,E2 -7400.129} C_VEL
LIN {X 0,Y 477.097,Z 717.455,A -85,B 0,C 180,E1 -7400.507,E2 -7400.507} C_VEL
LIN {X 0,Y 476.757,Z 730.259,A -85,B 0,C 180,E1 -7401.058,E2 -7401.058} C_VEL
LIN {X 0,Y 476.434,Z 741.728,A -85,B 0,C 180,E1 -7401.732,E2 -7401.732} C_VEL
LIN {X 0,Y 475.956,Z 752.996,A -85,B 0,C 180,E1 -7402.576,E2 -7402.576} C_VEL
LIN {X 0,Y 475.457,Z 763.773,A -85,B 0,C 180,E1 -7403.59,E2 -7403.59} C_VEL
LIN {X 0,Y 475.038,Z 773.224,A -85,B 0,C 180,E1 -7404.705,E2 -7404.705} C_VEL
LIN {X 0,Y 474.599,Z 781.489,A -85,B 0,C 180,E1 -7405.902,E2 -7405.902} C_VEL
LIN {X 0,Y 474.348,Z 789.003,A -85,B 0,C 180,E1 -7407.259,E2 -7407.259} C_VEL
LIN {X 0,Y 474.129,Z 795.037,A -85,B 0,C 180,E1 -7408.655,E2 -7408.655} C_VEL
LIN {X 0,Y 473.935,Z 800.335,A -85,B 0,C 180,E1 -7410.277,E2 -7410.277} C_VEL
LIN {X 0,Y 473.854,Z 802.71,A -85,B 0,C 180,E1 -7411.272,E2 -7411.272} C_VEL
LIN {X 0,Y 473.752,Z 804.556,A -85,B 0,C 180,E1 -7412.28,E2 -7412.28} C_VEL
LIN {X 0,Y 473.677,Z 806.213,A -85,B 0,C 180,E1 -7413.813,E2 -7413.813} C_VEL
LIN {X 0,Y 473.653,Z 806.569,A -85,B 0,C 180,E1 -7415.357,E2 -7415.357} C_VEL
LIN {X 0,Y 473.668,Z 805.774,A -85,B 0,C 180,E1 -7416.755,E2 -7416.755} C_VEL
LIN {X 0,Y 473.714,Z 803.884,A -85,B 0,C 180,E1 -7418.16,E2 -7418.16} C_VEL
LIN {X 0,Y 473.884,Z 800.71,A -85,B 0,C 180,E1 -7419.622,E2 -7419.622} C_VEL
LIN {X 0,Y 474.015,Z 796.915,A -85,B 0,C 180,E1 -7420.876,E2 -7420.876} C_VEL
LIN {X 0,Y 474.171,Z 791.836,A -85,B 0,C 180,E1 -7422.178,E2 -7422.178} C_VEL
LIN {X 0,Y 474.443,Z 785.514,A -85,B 0,C 180,E1 -7423.463,E2 -7423.463} C_VEL
LIN {X 0,Y 474.735,Z 777.795,A -85,B 0,C 180,E1 -7424.718,E2 -7424.718} C_VEL
LIN {X 0,Y 475.244,Z 768.219,A -85,B 0,C 180,E1 -7425.971,E2 -7425.971} C_VEL
LIN {X 0,Y 475.656,Z 758.468,A -85,B 0,C 180,E1 -7427,E2 -7427} C_VEL
LIN {X 0,Y 476.072,Z 748.043,A -85,B 0,C 180,E1 -7427.886,E2 -7427.886} C_VEL
LIN {X 0,Y 476.507,Z 736.585,A -85,B 0,C 180,E1 -7428.661,E2 -7428.661} C_VEL
LIN {X 0,Y 476.74,Z 730.943,A -85,B 0,C 180,E1 -7428.976,E2 -7428.976} C_VEL
LIN {X 0,Y 476.203,Z 727.366,A -85,B 0,C 180,E1 -7429.18,E2 -7429.18} C_VEL
LIN {X 0,Y 473.545,Z 721.806,A -85,B 0,C 180,E1 -7429.521,E2 -7429.521} C_VEL
LIN {X 0,Y 470.871,Z 716.122,A -85,B 0,C 180,E1 -7429.823,E2 -7429.823} C_VEL
LIN {X 0,Y 470.298,Z 712.356,A -85,B 0,C 180,E1 -7429.964,E2 -7429.964} C_VEL
LIN {X 0,Y 470.566,Z 699.389,A -85,B 0,C 180,E1 -7430.276,E2 -7430.276} C_VEL
LIN {X 0,Y 471.191,Z 610.458,A -85,B 0,C 180,E1 -7431.699,E2 -7431.699} C_VEL
LIN {X 0,Y 468.399,Z 597.205,A -85,B 0,C 180,E1 -7432.037,E2 -7432.037} C_VEL
LIN {X 0,Y 468.368,Z 591.391,A -85,B 0,C 180,E1 -7433.385,E2 -7433.385} C_VEL
LIN {X 0,Y 467.618,Z 587.238,A -85,B 0,C 180,E1 -7434.426,E2 -7434.426} C_VEL
LIN {X 0,Y 467.578,Z 587.239,A -85,B 0,C 180,E1 -7437.322,E2 -7437.322} C_VEL
LIN {X 0,Y 467.566,Z 587.239,A -85,B 0,C 180,E1 -7440.668,E2 -7440.668} C_VEL
LIN {X 0,Y 467.613,Z 587.232,A -85,B 0,C 180,E1 -7443.201,E2 -7443.201} C_VEL
LIN {X 0,Y 467.591,Z 587.238,A -85,B 0,C 180,E1 -7446.469,E2 -7446.469} C_VEL
LIN {X 0,Y 467.623,Z 587.234,A -85,B 0,C 180,E1 -7449.778,E2 -7449.778} C_VEL
LIN {X 0,Y 467.609,Z 587.237,A -85,B 0,C 180,E1 -7452.508,E2 -7452.508} C_VEL
LIN {X 0,Y 467.606,Z 587.233,A -85,B 0,C 180,E1 -7455.198,E2 -7455.198} C_VEL
LIN {X 0,Y 467.683,Z 587.226,A -85,B 0,C 180,E1 -7457.856,E2 -7457.856} C_VEL
LIN {X 0,Y 467.682,Z 587.223,A -85,B 0,C 180,E1 -7461.358,E2 -7461.358} C_VEL
LIN {X 0,Y 467.744,Z 587.218,A -85,B 0,C 180,E1 -7463.964,E2 -7463.964} C_VEL
LIN {X 0,Y 467.861,Z 587.201,A -85,B 0,C 180,E1 -7467.418,E2 -7467.418} C_VEL
LIN {X 0,Y 467.884,Z 587.2,A -85,B 0,C 180,E1 -7470.001,E2 -7470.001} C_VEL
LIN {X 0,Y 467.862,Z 587.21,A -85,B 0,C 180,E1 -7472.584,E2 -7472.584} C_VEL
LIN {X 0,Y 467.746,Z 587.217,A -85,B 0,C 180,E1 -7476.038,E2 -7476.038} C_VEL
LIN {X 0,Y 467.685,Z 587.231,A -85,B 0,C 180,E1 -7478.644,E2 -7478.644} C_VEL
LIN {X 0,Y 467.659,Z 587.227,A -85,B 0,C 180,E1 -7482.146,E2 -7482.146} C_VEL
LIN {X 0,Y 467.642,Z 587.228,A -85,B 0,C 180,E1 -7485.696,E2 -7485.696} C_VEL
LIN {X 0,Y 467.621,Z 587.238,A -85,B 0,C 180,E1 -7488.765,E2 -7488.765} C_VEL
LIN {X 0,Y 467.584,Z 587.24,A -85,B 0,C 180,E1 -7491.269,E2 -7491.269} C_VEL
LIN {X 0,Y 467.575,Z 587.237,A -85,B 0,C 180,E1 -7493.944,E2 -7493.944} C_VEL
LIN {X 0,Y 467.62,Z 587.236,A -85,B 0,C 180,E1 -7496.801,E2 -7496.801} C_VEL
LIN {X 0,Y 467.558,Z 587.24,A -85,B 0,C 180,E1 -7499.739,E2 -7499.739} C_VEL
LIN {X 0,Y 467.587,Z 587.238,A -85,B 0,C 180,E1 -7502.759,E2 -7502.759} C_VEL
LIN {X 0,Y 467.558,Z 587.24,A -85,B 0,C 180,E1 -7505.89,E2 -7505.89} C_VEL
LIN {X 0,Y 467.586,Z 587.242,A -85,B 0,C 180,E1 -7509.145,E2 -7509.145} C_VEL
LIN {X 0,Y 467.591,Z 587.235,A -85,B 0,C 180,E1 -7512.567,E2 -7512.567} C_VEL
LIN {X 0,Y 467.57,Z 587.241,A -85,B 0,C 180,E1 -7515.053,E2 -7515.053} C_VEL
LIN {X 0,Y 467.593,Z 587.243,A -85,B 0,C 180,E1 -7517.44,E2 -7517.44} C_VEL
LIN {X 0,Y 467.564,Z 587.239,A -85,B 0,C 180,E1 -7520.854,E2 -7520.854} C_VEL
LIN {X 0,Y 467.564,Z 587.239,A -85,B 0,C 180,E1 -7524.261,E2 -7524.261} C_VEL
LIN {X 0,Y 467.586,Z 587.24,A -85,B 0,C 180,E1 -7527.321,E2 -7527.321} C_VEL
LIN {X 0,Y 467.574,Z 587.237,A -85,B 0,C 180,E1 -7530.668,E2 -7530.668} C_VEL
LIN {X 0,Y 467.618,Z 587.233,A -85,B 0,C 180,E1 -7533.2,E2 -7533.2} C_VEL
LIN {X 0,Y 467.596,Z 587.235,A -85,B 0,C 180,E1 -7536.469,E2 -7536.469} C_VEL
LIN {X 0,Y 467.627,Z 587.238,A -85,B 0,C 180,E1 -7539.777,E2 -7539.777} C_VEL
LIN {X 0,Y 467.603,Z 587.234,A -85,B 0,C 180,E1 -7542.507,E2 -7542.507} C_VEL
LIN {X 0,Y 467.611,Z 587.233,A -85,B 0,C 180,E1 -7545.197,E2 -7545.197} C_VEL
LIN {X 0,Y 467.662,Z 587.233,A -85,B 0,C 180,E1 -7547.855,E2 -7547.855} C_VEL
